               // Sinal de andon do posto 6
           ELSIF #Out_LinhaEcu.Andons[5] THEN
               #Out_LinhaEcu.NumMensagem := 14;
               #Out_MensagemEcu := 'NECESSARIO AJUDA NO POSTO 6';

               // Sinal de andon do posto 7
           ELSIF #Out_LinhaEcu.Andons[6] THEN
               #Out_LinhaEcu.NumMensagem := 15;
               #Out_MensagemEcu := 'NECESSARIO AJUDA NO POSTO 7';

               // Sinal de andon do posto 8
           ELSIF #Out_LinhaEcu.Andons[7] THEN
               #Out_LinhaEcu.NumMensagem := 16;
               #Out_MensagemEcu := 'AGUARDANDO RETIRADA DO PRODUTO NO POSTO 8';

           END_IF;
           ;
           // Linha em parada de produção
       ELSIF #S_ForaDeTurno THEN
           #Out_LinhaEcu.NumMensagem := 17;
           #Out_MensagemEcu := 'LINHA EM PARADA DE PRODUÇÃO';

           // Verifica se o AGV está em modo manual
       ELSIF (#In_DadosEcu.Dados_Agv[0].AutomaticoManual = 1) OR
           (#In_DadosEcu.Dados_Agv[1].AutomaticoManual = 1) OR
           (#In_DadosEcu.Dados_Agv[2].AutomaticoManual = 1) OR
           (#In_DadosEcu.Dados_Agv[3].AutomaticoManual = 1) OR
             (#In_DadosEcu.Dados_Agv[4].AutomaticoManual = 1) OR
             (*(#In_DadosEcu.Dados_Agv[5].AutomaticoManual = 1) OR*)
           (#In_DadosEcu.Dados_Agv[6].AutomaticoManual = 1) OR 
           (#In_DadosEcu.Dados_Agv[7].AutomaticoManual = 1) THEN

           // Verifica se o AGV 1 está em modo manual e diz em qual posto
           IF (#In_DadosEcu.Dados_Agv[0].AutomaticoManual = 1) THEN
               #Out_LinhaEcu.NumMensagem := 18;
               #Out_MensagemEcu := CONCAT(IN1 := 'AGV 1 EM MODO MANUAL NO POSTO ', IN2 := INT_TO_STRING(#In_DadosEcu.Dados_Agv[0].Posto));

               // Verifica se o AGV 2 está em modo manual e diz em qual posto
           ELSIF (#In_DadosEcu.Dados_Agv[1].AutomaticoManual = 1) THEN
               #Out_LinhaEcu.NumMensagem := 19;
               #Out_MensagemEcu := CONCAT(IN1 := 'AGV 2  EM MODO MANUAL NO POSTO ', IN2 := INT_TO_STRING(#In_DadosEcu.Dados_Agv[1].Posto));

               // Verifica se o AGV 3 está em modo manual e diz em qual posto
           ELSIF (#In_DadosEcu.Dados_Agv[2].AutomaticoManual = 1) THEN
               #Out_LinhaEcu.NumMensagem := 20;
               #Out_MensagemEcu := CONCAT(IN1 := 'AGV 3 EM MODO MANUAL NO POSTO ', IN2 := INT_TO_STRING(#In_DadosEcu.Dados_Agv[2].Posto));

               // Verifica se o AGV 4 está em modo manual e diz em qual posto
           ELSIF (#In_DadosEcu.Dados_Agv[3].AutomaticoManual = 1) THEN
               #Out_LinhaEcu.NumMensagem := 21;
               #Out_MensagemEcu := CONCAT(IN1 := 'AGV 4 EM MODO MANUAL NO POSTO ', IN2 := INT_TO_STRING(#In_DadosEcu.Dados_Agv[3].Posto));

               // Verifica se o AGV 5 está em modo manual e diz em qual posto
           ELSIF (#In_DadosEcu.Dados_Agv[4].AutomaticoManual = 1 AND "AlwaysFALSE") THEN
               #Out_LinhaEcu.NumMensagem := 22;
               #Out_MensagemEcu := CONCAT(IN1 := 'AGV 5 EM MODO MANUAL NO POSTO ', IN2 := INT_TO_STRING(#In_DadosEcu.Dados_Agv[4].Posto));

               // Verifica se o AGV 6 está em modo manual e diz em qual posto
               (* ELSIF (#In_DadosEcu.Dados_Agv[5].AutomaticoManual = 1 AND "AlwaysFALSE") THEN
               #Out_LinhaEcu.NumMensagem := 23;
               #Out_MensagemEcu := CONCAT(IN1 := 'AGV 6 EM MODO MANUAL NO POSTO ', IN2 := INT_TO_STRING(#In_DadosEcu.Dados_Agv[5].Posto));
               *)
               // Verifica se o AGV 7 está em modo manual e diz em qual posto
           ELSIF (#In_DadosEcu.Dados_Agv[6].AutomaticoManual = 1) THEN
               #Out_LinhaEcu.NumMensagem := 24;
               #Out_MensagemEcu := CONCAT(IN1 := 'AGV 7 EM MODO MANUAL NO POSTO ', IN2 := INT_TO_STRING(#In_DadosEcu.Dados_Agv[6].Posto));

               // Verifica se o AGV 8 está em modo manual e diz em qual posto
           ELSIF (#In_DadosEcu.Dados_Agv[7].AutomaticoManual = 1) THEN
               #Out_LinhaEcu.NumMensagem := 25;
               #Out_MensagemEcu := CONCAT(IN1 := 'AGV8 EM MODO MANUAL NO POSTO ', IN2 := INT_TO_STRING(#In_DadosEcu.Dados_Agv[7].Posto));


           END_IF;


           //Verifica se algum AGV esta fora da rota
       ELSIF (#In_DadosEcu.Dados_Agv[0]."Erros.Agv"= 8) OR
           (#In_DadosEcu.Dados_Agv[1]."Erros.Agv" = 8) OR
           (#In_DadosEcu.Dados_Agv[2]."Erros.Agv" = 8) OR
           (#In_DadosEcu.Dados_Agv[3]."Erros.Agv" = 8) OR
           (#In_DadosEcu.Dados_Agv[4]."Erros.Agv" = 8 ) OR
           (#In_DadosEcu.Dados_Agv[5]."Erros.Agv" = 8 AND "AlwaysFALSE") OR
           (#In_DadosEcu.Dados_Agv[6]."Erros.Agv" = 8) OR
           (#In_DadosEcu.Dados_Agv[7]."Erros.Agv" = 8) THEN

           // Verifica se o AGV 1 está fora da rota
           IF (#In_DadosEcu.Dados_Agv[0]."Erros.Pgv" = 8) THEN
               #Out_LinhaEcu.NumMensagem := 26;
               #Out_MensagemEcu := CONCAT(IN1 := 'AGV 1 FORA DA ROTA NO POSTO ', IN2 := INT_TO_STRING(#In_DadosEcu.Dados_Agv[0].Posto));

               // Verifica se o AGV 2 está fora da rota
           ELSIF (#In_DadosEcu.Dados_Agv[1]."Erros.Agv" = 8) THEN
               #Out_LinhaEcu.NumMensagem := 27;
               #Out_MensagemEcu := CONCAT(IN1 := 'AGV 2 FORA DA ROTA NO POSTO ', IN2 := INT_TO_STRING(#In_DadosEcu.Dados_Agv[1].Posto));

               // Verifica se o AGV 3 está fora da rota
           ELSIF (#In_DadosEcu.Dados_Agv[2]."Erros.Agv" = 8) THEN
               #Out_LinhaEcu.NumMensagem := 28;
               #Out_MensagemEcu := CONCAT(IN1 := 'AGV 3 FORA DA ROTA NO POSTO ', IN2 := INT_TO_STRING(#In_DadosEcu.Dados_Agv[2].Posto));

               // Verifica se o AGV 4 está fora da rota
           ELSIF (#In_DadosEcu.Dados_Agv[3]."Erros.Agv" = 8) THEN
               #Out_LinhaEcu.NumMensagem := 29;
               #Out_MensagemEcu := CONCAT(IN1 := 'AGV 4 FORA DA ROTA NO POSTO ', IN2 := INT_TO_STRING(#In_DadosEcu.Dados_Agv[3].Posto));

               // Verifica se o AGV 5 está fora da rota
           ELSIF (#In_DadosEcu.Dados_Agv[4]."Erros.Agv" = 8 AND "AlwaysFALSE") THEN
               #Out_LinhaEcu.NumMensagem := 30;
               #Out_MensagemEcu := CONCAT(IN1 := 'AGV 5 FORA DA ROTA NO POSTO ', IN2 := INT_TO_STRING(#In_DadosEcu.Dados_Agv[4].Posto));

               // Verifica se o AGV 6 está fora da rota
           ELSIF (#In_DadosEcu.Dados_Agv[5]."Erros.Agv" = 8 AND "AlwaysFALSE") THEN
               #Out_LinhaEcu.NumMensagem := 31;
               #Out_MensagemEcu := CONCAT(IN1 := 'AGV 6 FORA DA ROTA NO POSTO ', IN2 := INT_TO_STRING(#In_DadosEcu.Dados_Agv[5].Posto));
               // Verifica se o AGV 7 está fora da rota
           ELSIF (#In_DadosEcu.Dados_Agv[6]."Erros.Agv" = 8) THEN
               #Out_LinhaEcu.NumMensagem := 32;
               #Out_MensagemEcu := CONCAT(IN1 := 'AGV 7 FORA DA ROTA NO POSTO ', IN2 := INT_TO_STRING(#In_DadosEcu.Dados_Agv[6].Posto));
               // Verifica se o AGV 8 está fora da rota
           ELSIF (#In_DadosEcu.Dados_Agv[7]."Erros.Agv" = 8) THEN
               #Out_LinhaEcu.NumMensagem := 33;
               #Out_MensagemEcu := CONCAT(IN1 := 'AGV 8 FORA DA ROTA NO POSTO ', IN2 := INT_TO_STRING(#In_DadosEcu.Dados_Agv[7].Posto));


           END_IF; 

       ELSE
           #Out_LinhaEcu.NumMensagem := 0;
           #Out_MensagemEcu := 'LINHA LIBERADA';
       END_IF;

   END_REGION

   // Coloca os dados das memorias nas saidas do bloco
   REGION Saidas
       // Coloca os dados das memorias nas saidas do bloco
       #Out_LinhaEcu.Tempo_Takt := #In_DadosEcu.Dados_Takt.Tempo_Takt;
       #Out_LinhaEcu.Tempo_StopTime := #In_DadosEcu.Dados_Takt.Tempo_StopTime;
       #Out_LinhaEcu.Objetivo := #In_DadosEcu.Dados_Takt.Objetivo;
       #Out_LinhaEcu.Atual := #In_DadosEcu.Dados_Takt.Atual;
       #Out_LinhaEcu.DirectRun := 99.9;
       #Out_LinhaEcu.LinhaParada := #S_ForaDeTurno;
       #Out_LinhaEcu.TempoRetornoParada := #S_TempoRetorno;
       #Out_LinhaEcu.LinhaRodando := NOT #S_ForaDeTurno;
   END_REGION
END_FUNCTION_BLOCK

FUNCTION_BLOCK "FB203_FiltroDados_Skd"   // FB203, SCL
TITLE = FB203_FiltroDados_Skd
{ S7_Optimized_Access := 'TRUE' }
VERSION : 0.1
// FB203_FiltroDados_Skd
   VAR_INPUT
      In_InfoCabinas : "TAKT_OUTPUT.INFORMATION";
      In_Turno : Struct
         Turnos : Array[0..2] of Struct
            Inicio : Date_And_Time;
            Fim : Date_And_Time;
            Objetivo : Int;
            DiasDaSemana : Array[0..6] of Bool;
            Paradas : Array[0..5] of Struct
               Inicio : Date_And_Time;
               Fim : Date_And_Time;
            END_STRUCT;
            HE_Inicio : Date_And_Time;
            HE_Fim : Date_And_Time;
         END_STRUCT;
      END_STRUCT;
   END_VAR
   VAR_OUTPUT
      Out_Linha : Struct
         Tempo_Takt : DInt;
         Tempo_StopTime : DInt;
         Objetivo : Int;
         Atual : Int;
         LinhaParada : Bool;
         TempoRetornoParada : DInt;
         LinhaRodando : Bool;
         Andons : Array[0..8] of Bool;
         CorDeTela : Byte;
         DirectRun : Real;
         SaldoDoTurno : Int;
         AndonOn : Int;
         Paradas : Array[0..1] of Struct
            Inicio : Time_Of_Day;
            Fim : Time_Of_Day;
            Posto : Int;
            ValorTimer : Int;
            ValorTimerFim : Int;
         END_STRUCT;
         NumMensagem : Int;
         Emergencias : Array[0..8] of Bool;
      END_STRUCT;
      Out_Mensagem : String;
   END_VAR
   VAR
      S_DateTime : Date_And_Time;
      S_CounterFor : Int;
      S_CounterFor_1 : Int;
      S_Turnos : Array[0..2] of Struct
         Paradas : Array[0..6] of Bool;
         ContagemRetorno : Array[0..6] of DInt;
      END_STRUCT;
      S_ForaDeTurno : Bool;
      S_TempoRetorno : DInt;
      S_Hora : Time_Of_Day;
   END_VAR
   VAR_TEMP
      Err : Int;
   END_VAR
BEGIN
   (*
       ESTE BLOCO REALIZA O FILTRO DAS INFORMAÇÕES DO TAKT, EXEMPLOS: TROCA DA COR DA TELA, MENSAGENS NA TELA E ETC
   *)


   // Converte o sinal de andon de byte para boolean
   REGION Valores ANDON
       // Converte o sinal de andon de byte para boolean
       #Out_Linha.Andons[0] := #In_InfoCabinas.ANDON.%X0;
       #Out_Linha.Andons[1] := #In_InfoCabinas.ANDON.%X1;
       #Out_Linha.Andons[2] := #In_InfoCabinas.ANDON.%X2;
       #Out_Linha.Andons[3] := #In_InfoCabinas.ANDON.%X3;
       #Out_Linha.Andons[4] := #In_InfoCabinas.ANDON.%X4;
       #Out_Linha.Andons[5] := #In_InfoCabinas.ANDON.%X5;
       #Out_Linha.Andons[6] := #In_InfoCabinas.ANDON.%X6;
       #Out_Linha.Andons[7] := #In_InfoCabinas.ANDON.%X7;
   END_REGION

   // Converte o sinal de emergencia de byte para boolean
   REGION Valores Emergencia
       // Converte o sinal de emergencia de byte para boolean
       #Out_Linha.Emergencias[0] := #In_InfoCabinas.EMERGENCY.%X0;
       #Out_Linha.Emergencias[1] := #In_InfoCabinas.EMERGENCY.%X1;
       #Out_Linha.Emergencias[2] := #In_InfoCabinas.EMERGENCY.%X2;
       #Out_Linha.Emergencias[3] := #In_InfoCabinas.EMERGENCY.%X3;
       #Out_Linha.Emergencias[4] := #In_InfoCabinas.EMERGENCY.%X4;
       #Out_Linha.Emergencias[5] := #In_InfoCabinas.EMERGENCY.%X5;
       #Out_Linha.Emergencias[6] := #In_InfoCabinas.EMERGENCY.%X6;
       #Out_Linha.Emergencias[7] := #In_InfoCabinas.EMERGENCY.%X7;
   END_REGION

   //Realiza a leitura da hora atual do CLP
   REGION HoraAtual

       //Realiza a leitura da hora atual do CLP
       #Err := RD_LOC_T(#S_DateTime);

   END_REGION
   REGION VerificaEmTurno
       #S_Hora := DT_TO_TOD(#S_DateTime);
       IF #S_Hora > TOD#16:00:00 THEN
           #S_TempoRetorno := TOD_TO_DINT(TOD#07:00:00) - TOD_TO_DINT(#S_Hora);
           #S_ForaDeTurno := 1;
       ELSE
           #S_TempoRetorno := 0;
           #S_ForaDeTurno := 0;
       END_IF;


   END_REGION
   //Verifica se a linha esta em turno, caso não esteja retorno o tempo necessario para a linha voltar a rodar
   REGION LinhaEmTurno
       FOR #S_CounterFor := 0 TO 2 DO
           //Verifica se está em turno
           IF #In_Turno.Turnos[#S_CounterFor].Inicio >= #S_DateTime AND #S_DateTime <= #In_Turno.Turnos[#S_CounterFor].Fim THEN
               //Verifica se existe alguma parada programada
               FOR #S_CounterFor_1 := 0 TO 5 DO
                   IF #In_Turno.Turnos[#S_CounterFor].Paradas[#S_CounterFor_1].Inicio >= #S_DateTime
                       AND #S_DateTime <= #In_Turno.Turnos[#S_CounterFor].Paradas[#S_CounterFor_1].Fim THEN

                       #S_Turnos[#S_CounterFor].Paradas[#S_CounterFor_1] := 1;
                       #S_Turnos[#S_CounterFor].ContagemRetorno[#S_CounterFor_1] := TOD_TO_DINT(DT_TO_TOD(#S_DateTime - (#In_Turno.Turnos[#S_CounterFor].Paradas[#S_CounterFor_1].Fim - #In_Turno.Turnos[#S_CounterFor].Paradas[#S_CounterFor_1].Inicio)));
                   ELSE
                       #S_Turnos[#S_CounterFor].ContagemRetorno[#S_CounterFor_1] := 0;
                       #S_Turnos[#S_CounterFor].Paradas[#S_CounterFor_1] := 0;

                   END_IF;

                   #S_Turnos[#S_CounterFor].Paradas[6] := 0; // Em turno
                   #S_Turnos[#S_CounterFor].ContagemRetorno[6] := 0;
               END_FOR;
           ELSE
               #S_Turnos[#S_CounterFor].Paradas[6] := 1; // Fora de turno
               #S_Turnos[#S_CounterFor].ContagemRetorno[6] := #S_DateTime - #In_Turno.Turnos[#S_CounterFor].Paradas[#S_CounterFor_1].Inicio; // Quantidade de tempo restante para reiniciar o novo turno
           END_IF;

       END_FOR;

       #S_ForaDeTurno := #S_Turnos[0 AND 1 AND 2].Paradas[0 AND 1 AND 2 AND 3 AND 4 AND 5 AND 6];
       #S_TempoRetorno := #S_Turnos[0 AND 1 AND 2].ContagemRetorno[0 AND 1 AND 2 AND 3 AND 4 AND 5 AND 6];
   END_REGION

   // Realiza a analise de todos os dados e troca a cor da tela
   REGION DefiniçãoCorDaTela
       // 1 - Tela Amarela (Necessario ajuda em algum posto e não estourou o tempo do TAKT)
       IF ((#Out_Linha.Andons[1] OR #Out_Linha.Andons[3] OR #Out_Linha.Andons[4] OR #Out_Linha.Andons[6] OR #Out_Linha.Andons[7]) AND (#In_InfoCabinas.TAKT_ET > 0) AND NOT #S_ForaDeTurno) THEN
           #Out_Linha.CorDeTela := 1;

           // 2 - Tela Vermelho (Necessario ajuda em algum posto e estourou o tempo do TAKT)
       ELSIF (((#Out_Linha.Andons[0] OR #Out_Linha.Andons[1] OR #Out_Linha.Andons[3] OR #Out_Linha.Andons[4] OR #Out_Linha.Andons[6] OR #Out_Linha.Andons[7]) AND (#In_InfoCabinas.TAKT_ET = 0)) OR (#In_InfoCabinas.EMERGENCY <> 0)) AND NOT #S_ForaDeTurno THEN
           #Out_Linha.CorDeTela := 2;

           //3 - Tela Azul - (Aguardando inicio de turno/Volta da refeição)
       ELSIF #S_ForaDeTurno THEN
           #Out_Linha.CorDeTela := 3;

           //4 - Tela Laranja - (Aguardando retirada do produto)
       ELSIF ((#Out_Linha.Andons[0] OR #Out_Linha.Andons[7])) AND NOT #S_ForaDeTurno THEN
           #Out_Linha.CorDeTela := 4;
           //0 - Tela Branca/Preta (Tudo Ok)
       ELSE
           #Out_Linha.CorDeTela := 0;
       END_IF;


   END_REGION

   // Realiza a analise de todos os dados e escreve a mensagem na tela 
   REGION Mensagens

       IF #In_InfoCabinas.EMERGENCY <> 0 AND NOT #S_ForaDeTurno THEN

           // Sinal de EMERGÊNCIA  do posto 1
           IF #Out_Linha.Emergencias[0] THEN
               #Out_Linha.NumMensagem := 1;
               #Out_Mensagem := 'EMERGÊNCIA  ACIONADO NO POSTO 1';

               // Sinal de EMERGÊNCIA  do posto 2
           ELSIF #Out_Linha.Emergencias[1] THEN
               #Out_Linha.NumMensagem := 2;
               #Out_Mensagem := 'EMERGÊNCIA  ACIONADO NO POSTO 2';

               // Sinal de EMERGÊNCIA  do posto 3
           ELSIF #Out_Linha.Emergencias[2] THEN
               #Out_Linha.NumMensagem := 3;
               #Out_Mensagem := 'EMERGÊNCIA  ACIONADO NO POSTO 3';

               // Sinal de EMERGÊNCIA  do posto 4
           ELSIF #Out_Linha.Emergencias[3] THEN
               #Out_Linha.NumMensagem := 4;
               #Out_Mensagem := 'EMERGÊNCIA  ACIONADO NO POSTO 4';

               // Sinal de EMERGÊNCIA  do posto 5
           ELSIF #Out_Linha.Emergencias[4] THEN
               #Out_Linha.NumMensagem := 5;
               #Out_Mensagem := 'EMERGÊNCIA  ACIONADO NO POSTO 5';

               // Sinal de EMERGÊNCIA  do posto 6
           ELSIF #Out_Linha.Emergencias[5] THEN
               #Out_Linha.NumMensagem := 6;
               #Out_Mensagem := 'EMERGÊNCIA  ACIONADO NO POSTO 6';

               // Sinal de EMERGÊNCIA  do posto 7
           ELSIF #Out_Linha.Emergencias[6] THEN
               #Out_Linha.NumMensagem := 7;
               #Out_Mensagem := 'EMERGÊNCIA  ACIONADO NO POSTO 7';

               // Sinal de EMERGÊNCIA  do posto 8
           ELSIF #Out_Linha.Emergencias[7] THEN
               #Out_Linha.NumMensagem := 8;
               #Out_Mensagem := 'EMERGÊNCIA  ACIONADO NO POSTO 8';

           END_IF;

       ELSIF #In_InfoCabinas.ANDON <> 0 AND NOT #S_ForaDeTurno THEN

           // Sinal de andon do posto 1
           IF #Out_Linha.Andons[0] THEN
               #Out_Linha.NumMensagem := 9;
               #Out_Mensagem := 'NECESSARIO AJUDA NO POSTO 1';

               // Sinal de andon do posto 2
           ELSIF #Out_Linha.Andons[1] THEN
               #Out_Linha.NumMensagem := 10;
               #Out_Mensagem := 'NECESSARIO AJUDA NO POSTO 2';

               // Sinal de andon do posto 3
           ELSIF #Out_Linha.Andons[2] THEN
               #Out_Linha.NumMensagem := 11;
               #Out_Mensagem := 'NECESSARIO AJUDA NO POSTO 3';

               // Sinal de andon do posto 4
           ELSIF #Out_Linha.Andons[3] THEN
               #Out_Linha.NumMensagem := 12;
               #Out_Mensagem := 'NECESSARIO AJUDA NO POSTO 4';

               // Sinal de andon do posto 5
           ELSIF #Out_Linha.Andons[4] THEN
               #Out_Linha.NumMensagem := 13;
               #Out_Mensagem := 'NECESSARIO AJUDA NO POSTO 5';

               // Sinal de andon do posto 6
           ELSIF #Out_Linha.Andons[5] THEN
               #Out_Linha.NumMensagem := 14;
               #Out_Mensagem := 'NECESSARIO AJUDA NO POSTO 6';

               // Sinal de andon do posto 7
           ELSIF #Out_Linha.Andons[6] THEN
               #Out_Linha.NumMensagem := 15;
               #Out_Mensagem := 'NECESSARIO AJUDA NO POSTO 7';

               // Sinal de andon do posto 8
           ELSIF #Out_Linha.Andons[7] THEN
               #Out_Linha.NumMensagem := 16;
               #Out_Mensagem := 'NECESSARIO AJUDA NO POSTO 8';

           END_IF;
           ;
           // Linha em parada de produção
       ELSIF #S_ForaDeTurno THEN
           #Out_Linha.NumMensagem := 17;
           #Out_Mensagem := 'LINHA EM PARADA DE PRODUÇÃO';
       ELSE
           #Out_Linha.NumMensagem := 0;
           #Out_Mensagem := 'LINHA LIBERADA';
       END_IF;

   END_REGION

   // Coloca os dados das memorias nas saidas do bloco
   REGION Saidas
       // Coloca os dados das memorias nas saidas do bloco
       #Out_Linha.Tempo_Takt := #In_InfoCabinas.TAKT_ET;
       #Out_Linha.Tempo_StopTime := #In_InfoCabinas.STOP_TIME;
       #Out_Linha.Objetivo := #In_InfoCabinas.TARGET;
       #Out_Linha.Atual := #In_InfoCabinas.ACTUAL_PRODUCTION;
       #Out_Linha.DirectRun := 99.9;
       #Out_Linha.LinhaParada := #S_ForaDeTurno;
       #Out_Linha.TempoRetornoParada := #S_TempoRetorno;
       #Out_Linha.LinhaRodando := NOT #S_ForaDeTurno;
   END_REGION
END_FUNCTION_BLOCK

FUNCTION_BLOCK "FB204_FiltroDados_Comp"   // FB204, SCL
TITLE = FB204_FiltroDados_Comp
{ S7_Optimized_Access := 'TRUE' }
VERSION : 0.1
// FB204_FiltroDados_Comp
   VAR_INPUT
      In_InfoCabinas : "TAKT_OUTPUT.INFORMATION";
      In_Turno : Struct
         Turnos : Array[0..2] of Struct
            Inicio : Date_And_Time;
            Fim : Date_And_Time;
            Objetivo : Int;
            DiasDaSemana : Array[0..6] of Bool;
            Paradas : Array[0..5] of Struct
               Inicio : Date_And_Time;
               Fim : Date_And_Time;
            END_STRUCT;
            HE_Inicio : Date_And_Time;
            HE_Fim : Date_And_Time;
         END_STRUCT;
      END_STRUCT;
   END_VAR
   VAR_OUTPUT
      Out_Linha : Struct
         Tempo_Takt : DInt;
         Tempo_StopTime : DInt;
         Objetivo : Int;
         Atual : Int;
         LinhaParada : Bool;
         TempoRetornoParada : DInt;
         LinhaRodando : Bool;
         Andons : Array[0..8] of Bool;
         CorDeTela : Byte;
         DirectRun : Real;
         SaldoDoTurno : Int;
         AndonOn : Int;
         Paradas : Array[0..1] of Struct
            Inicio : Time_Of_Day;
            Fim : Time_Of_Day;
            Posto : Int;
            ValorTimer : Int;
            ValorTimerFim : Int;
         END_STRUCT;
         NumMensagem : Int;
         Emergencias : Array[0..8] of Bool;
      END_STRUCT;
      Out_Mensagem : String;
   END_VAR
   VAR
      S_DateTime : Date_And_Time;
      S_CounterFor : Int;
      S_CounterFor_1 : Int;
      S_Turnos : Array[0..2] of Struct
         Paradas : Array[0..6] of Bool;
         ContagemRetorno : Array[0..6] of DInt;
      END_STRUCT;
      S_ForaDeTurno : Bool;
      S_TempoRetorno : DInt;
      S_Hora : Time_Of_Day;
   END_VAR
   VAR_TEMP
      Err : Int;
   END_VAR
BEGIN
   (*
       ESTE BLOCO REALIZA O FILTRO DAS INFORMAÇÕES DO TAKT, EXEMPLOS: TROCA DA COR DA TELA, MENSAGENS NA TELA E ETC
   *)


   // Converte o sinal de andon de byte para boolean
   REGION Valores ANDON
       // Converte o sinal de andon de byte para boolean
       #Out_Linha.Andons[0] := #In_InfoCabinas.ANDON.%X0;
       #Out_Linha.Andons[1] := #In_InfoCabinas.ANDON.%X1;
       #Out_Linha.Andons[2] := #In_InfoCabinas.ANDON.%X2;
       #Out_Linha.Andons[3] := #In_InfoCabinas.ANDON.%X3;
       #Out_Linha.Andons[4] := #In_InfoCabinas.ANDON.%X4;
       #Out_Linha.Andons[5] := #In_InfoCabinas.ANDON.%X5;
       #Out_Linha.Andons[6] := #In_InfoCabinas.ANDON.%X6;
       #Out_Linha.Andons[7] := #In_InfoCabinas.ANDON.%X7;
   END_REGION

   // Converte o sinal de emergencia de byte para boolean
   REGION Valores Emergencia
       // Converte o sinal de emergencia de byte para boolean
       #Out_Linha.Emergencias[0] := #In_InfoCabinas.EMERGENCY.%X0;
       #Out_Linha.Emergencias[1] := #In_InfoCabinas.EMERGENCY.%X1;
       #Out_Linha.Emergencias[2] := #In_InfoCabinas.EMERGENCY.%X2;
       #Out_Linha.Emergencias[3] := #In_InfoCabinas.EMERGENCY.%X3;
       #Out_Linha.Emergencias[4] := #In_InfoCabinas.EMERGENCY.%X4;
       #Out_Linha.Emergencias[5] := #In_InfoCabinas.EMERGENCY.%X5;
       #Out_Linha.Emergencias[6] := #In_InfoCabinas.EMERGENCY.%X6;
       #Out_Linha.Emergencias[7] := #In_InfoCabinas.EMERGENCY.%X7;
   END_REGION

   //Realiza a leitura da hora atual do CLP
   REGION HoraAtual

       //Realiza a leitura da hora atual do CLP
       #Err := RD_LOC_T(#S_DateTime);

   END_REGION
   REGION VerificaEmTurno
       #S_Hora := DT_TO_TOD(#S_DateTime);
       IF #S_Hora > TOD#16:00:00 THEN
           #S_TempoRetorno := TOD_TO_DINT(TOD#07:00:00) - TOD_TO_DINT(#S_Hora);
           #S_ForaDeTurno := 1;
       ELSE
           #S_TempoRetorno := 0;
           #S_ForaDeTurno := 0;
       END_IF;


   END_REGION
   //Verifica se a linha esta em turno, caso não esteja retorno o tempo necessario para a linha voltar a rodar
   REGION LinhaEmTurno
       FOR #S_CounterFor := 0 TO 2 DO
           //Verifica se está em turno
           IF #In_Turno.Turnos[#S_CounterFor].Inicio >= #S_DateTime AND #S_DateTime <= #In_Turno.Turnos[#S_CounterFor].Fim THEN
               //Verifica se existe alguma parada programada
               FOR #S_CounterFor_1 := 0 TO 5 DO
                   IF #In_Turno.Turnos[#S_CounterFor].Paradas[#S_CounterFor_1].Inicio >= #S_DateTime
                       AND #S_DateTime <= #In_Turno.Turnos[#S_CounterFor].Paradas[#S_CounterFor_1].Fim THEN

                       #S_Turnos[#S_CounterFor].Paradas[#S_CounterFor_1] := 1;
                       #S_Turnos[#S_CounterFor].ContagemRetorno[#S_CounterFor_1] := TOD_TO_DINT(DT_TO_TOD(#S_DateTime - (#In_Turno.Turnos[#S_CounterFor].Paradas[#S_CounterFor_1].Fim - #In_Turno.Turnos[#S_CounterFor].Paradas[#S_CounterFor_1].Inicio)));
                   ELSE
                       #S_Turnos[#S_CounterFor].ContagemRetorno[#S_CounterFor_1] := 0;
                       #S_Turnos[#S_CounterFor].Paradas[#S_CounterFor_1] := 0;

                   END_IF;

                   #S_Turnos[#S_CounterFor].Paradas[6] := 0; // Em turno
                   #S_Turnos[#S_CounterFor].ContagemRetorno[6] := 0;
               END_FOR;
           ELSE
               #S_Turnos[#S_CounterFor].Paradas[6] := 1; // Fora de turno
               #S_Turnos[#S_CounterFor].ContagemRetorno[6] := #S_DateTime - #In_Turno.Turnos[#S_CounterFor].Paradas[#S_CounterFor_1].Inicio; // Quantidade de tempo restante para reiniciar o novo turno
           END_IF;

       END_FOR;

       #S_ForaDeTurno := #S_Turnos[0 AND 1 AND 2].Paradas[0 AND 1 AND 2 AND 3 AND 4 AND 5 AND 6];
       #S_TempoRetorno := #S_Turnos[0 AND 1 AND 2].ContagemRetorno[0 AND 1 AND 2 AND 3 AND 4 AND 5 AND 6];
   END_REGION

   // Realiza a analise de todos os dados e troca a cor da tela
   REGION DefiniçãoCorDaTela
       // 1 - Tela Amarela (Necessario ajuda em algum posto e não estourou o tempo do TAKT)
       IF (( #Out_Linha.Andons[1] OR #Out_Linha.Andons[3] OR #Out_Linha.Andons[5] OR #Out_Linha.Andons[7]) AND (#In_InfoCabinas.TAKT_ET > 0)) AND NOT #S_ForaDeTurno THEN
           #Out_Linha.CorDeTela := 1;

           // 2 - Tela Vermelho (Necessario ajuda em algum posto e estourou o tempo do TAKT)
       ELSIF ((( #Out_Linha.Andons[1] OR #Out_Linha.Andons[3] OR #Out_Linha.Andons[5] OR #Out_Linha.Andons[7]) AND (#In_InfoCabinas.TAKT_ET <= 0)) OR (#In_InfoCabinas.EMERGENCY <> 0)) AND NOT #S_ForaDeTurno THEN
           #Out_Linha.CorDeTela := 2;

           //3 - Tela Azul - (Aguardando inicio de turno/Volta da refeição)
       ELSIF #S_ForaDeTurno THEN
           #Out_Linha.CorDeTela := 3;

           //4 - Tela Laranja - (Aguardando retirada do produto)
       ELSIF ((#Out_Linha.Andons[0] OR #Out_Linha.Andons[4])) AND NOT #S_ForaDeTurno THEN
           #Out_Linha.CorDeTela := 4;
           //0 - Tela Branca/Preta (Tudo Ok)
       ELSE
           #Out_Linha.CorDeTela := 0;
       END_IF;


   END_REGION

   // Realiza a analise de todos os dados e escreve a mensagem na tela 
   REGION Mensagens

       IF #In_InfoCabinas.EMERGENCY <> 0 AND NOT #S_ForaDeTurno THEN

           // Sinal de EMERGÊNCIA  do posto 1
           IF #Out_Linha.Emergencias[0] THEN
               #Out_Linha.NumMensagem := 1;
               #Out_Mensagem := 'EMERGÊNCIA  ACIONADO NO POSTO 1';

               // Sinal de EMERGÊNCIA  do posto 2
           ELSIF #Out_Linha.Emergencias[1] THEN
               #Out_Linha.NumMensagem := 2;
               #Out_Mensagem := 'EMERGÊNCIA  ACIONADO NO POSTO 2';

               // Sinal de EMERGÊNCIA  do posto 3
           ELSIF #Out_Linha.Emergencias[2] THEN
               #Out_Linha.NumMensagem := 3;
               #Out_Mensagem := 'EMERGÊNCIA  ACIONADO NO POSTO 3';

               // Sinal de EMERGÊNCIA  do posto 4
           ELSIF #Out_Linha.Emergencias[3] THEN
               #Out_Linha.NumMensagem := 4;
               #Out_Mensagem := 'EMERGÊNCIA  ACIONADO NO POSTO 4';

               // Sinal de EMERGÊNCIA  do posto 5
           ELSIF #Out_Linha.Emergencias[4] THEN
               #Out_Linha.NumMensagem := 5;
               #Out_Mensagem := 'EMERGÊNCIA  ACIONADO NO POSTO 5';

               // Sinal de EMERGÊNCIA  do posto 6
           ELSIF #Out_Linha.Emergencias[5] THEN
               #Out_Linha.NumMensagem := 6;
               #Out_Mensagem := 'EMERGÊNCIA  ACIONADO NO POSTO 6';

               // Sinal de EMERGÊNCIA  do posto 7
           ELSIF #Out_Linha.Emergencias[6] THEN
               #Out_Linha.NumMensagem := 7;
               #Out_Mensagem := 'EMERGÊNCIA  ACIONADO NO POSTO 7';

               // Sinal de EMERGÊNCIA  do posto 8
           ELSIF #Out_Linha.Emergencias[7] THEN
               #Out_Linha.NumMensagem := 8;
               #Out_Mensagem := 'EMERGÊNCIA  ACIONADO NO POSTO 8';

           END_IF;

       ELSIF #In_InfoCabinas.ANDON <> 0 AND NOT #S_ForaDeTurno THEN

           // Sinal de andon do posto 1
           IF #Out_Linha.Andons[0] THEN
               #Out_Linha.NumMensagem := 9;
               #Out_Mensagem := 'NECESSARIO AJUDA NO POSTO 1';

               // Sinal de andon do posto 2
           ELSIF #Out_Linha.Andons[1] THEN
               #Out_Linha.NumMensagem := 10;
               #Out_Mensagem := 'NECESSARIO AJUDA NO POSTO 2';

               // Sinal de andon do posto 3
           ELSIF #Out_Linha.Andons[2] THEN
               #Out_Linha.NumMensagem := 11;
               #Out_Mensagem := 'NECESSARIO AJUDA NO POSTO 3';

               // Sinal de andon do posto 4
           ELSIF #Out_Linha.Andons[3] THEN
               #Out_Linha.NumMensagem := 12;
               #Out_Mensagem := 'NECESSARIO AJUDA NO POSTO 4';

               // Sinal de andon do posto 5
           ELSIF #Out_Linha.Andons[4] THEN
               #Out_Linha.NumMensagem := 13;
               #Out_Mensagem := 'AGUARDANDO RETIRADA DO PRODUTO NO POSTO 5';

               // Sinal de andon do posto 6
           ELSIF #Out_Linha.Andons[5] THEN
               #Out_Linha.NumMensagem := 14;
               #Out_Mensagem := 'NECESSARIO AJUDA NO POSTO 6';

               // Sinal de andon do posto 7
           ELSIF #Out_Linha.Andons[6] THEN
               #Out_Linha.NumMensagem := 15;
               #Out_Mensagem := 'NECESSARIO AJUDA NO POSTO 7';

               // Sinal de andon do posto 8
           ELSIF #Out_Linha.Andons[7] THEN
               #Out_Linha.NumMensagem := 16;
               #Out_Mensagem := 'NECESSARIO AJUDA NO POSTO 8';

           END_IF;
           ;
           // Linha em parada de produção
       ELSIF #S_ForaDeTurno THEN
           #Out_Linha.NumMensagem := 17;
           #Out_Mensagem := 'LINHA EM PARADA DE PRODUÇÃO';
       ELSE
           #Out_Linha.NumMensagem := 0;
           #Out_Mensagem := 'LINHA LIBERADA';
       END_IF;

   END_REGION

   // Coloca os dados das memorias nas saidas do bloco
   REGION Saidas
       // Coloca os dados das memorias nas saidas do bloco
       #Out_Linha.Tempo_Takt := #In_InfoCabinas.TAKT_ET;
       #Out_Linha.Tempo_StopTime := #In_InfoCabinas.STOP_TIME;
      #Out_Linha.Objetivo := #In_InfoCabinas.TARGET;
       #Out_Linha.Atual := #In_InfoCabinas.ACTUAL_PRODUCTION;
       #Out_Linha.DirectRun := 99.9;
       #Out_Linha.LinhaParada := #S_ForaDeTurno;
       #Out_Linha.TempoRetornoParada := #S_TempoRetorno;
       #Out_Linha.LinhaRodando := NOT #S_ForaDeTurno;
   END_REGION
END_FUNCTION_BLOCK

FUNCTION_BLOCK "FB205_FiltroDadosAgv"   // FB205, SCL
TITLE = FB205_FiltroDadosAgv
{ S7_Optimized_Access := 'TRUE' }
VERSION : 0.1
// FB205_FiltroDadosAgvs
   VAR_INPUT
      In : "Agv.Database";
   END_VAR
   VAR_OUTPUT
      Out_Sinais : Byte;
      Out_Posto : Byte;
      Out_Comando : Byte;
      Out_Velocidade : Byte;
      Out_Processo : Byte;
      Out_VelAtual : Byte;
      "Out_Erros.Agv" : Byte;
      "Out_Erros.Pgv" : Byte;
      "Out_Erros.MotorPasso" : Byte;
   END_VAR
BEGIN



   //#In_InfoCabinas.ANDON.%X0;
   IF #In.Emergencia THEN
       #Out_Sinais.%X0 := 1;
   ELSE
       #Out_Sinais.%X0 := 0;
   END_IF;

   IF #In.Safety THEN
       #Out_Sinais.%X1 := 1;
   ELSE
       #Out_Sinais.%X1 := 0;
   END_IF;

   IF #In.Warning THEN
       #Out_Sinais.%X2 := 1;
   ELSE
       #Out_Sinais.%X2 := 0;
   END_IF;

   IF #In.Rodando THEN
       #Out_Sinais.%X3 := 1;
   ELSE
       #Out_Sinais.%X3 := 0;
   END_IF;


   IF #In.AutomaticoManual = 2 THEN
       #Out_Sinais.%X4 := 1;
   ELSE
       #Out_Sinais.%X4 := 0;
   END_IF;

   IF #In.ConectarTakt  THEN
       #Out_Sinais.%X5 := 1;
   ELSE
       #Out_Sinais.%X5 := 0;
   END_IF;

   IF #In.Falha  THEN
       #Out_Sinais.%X6 := 1;
   ELSE
       #Out_Sinais.%X6 := 0;
   END_IF;

   IF #In.AutomaticoManual = 1 THEN
       #Out_Sinais.%X7 := 1;
   ELSE
       #Out_Sinais.%X7 := 0;
   END_IF;



   #Out_Posto := #In.Posto;
   #Out_Comando := #In.Comando;
   #Out_Velocidade := #In.Velocidade;
   #Out_Processo := #In.Processo;
   #Out_VelAtual := INT_TO_BYTE((#In.VelocidadeAtual/1000));
   #"Out_Erros.Agv" := #In."Erros.Agv";
   #"Out_Erros.Pgv" := #In."Erros.Pgv";
   #"Out_Erros.MotorPasso" := #In."Erros.Rfid";
END_FUNCTION_BLOCK

FUNCTION_BLOCK "FB206_CheckEmTurno"   // FB206, SCL
TITLE = FB206_EmTurno
{ S7_Optimized_Access := 'TRUE' }
VERSION : 0.1
   VAR_INPUT
      In_Turnos : Array[0..2] of Struct
         Inicio : Date_And_Time;
         Fim : Date_And_Time;
      END_STRUCT;
      In_Paradas : Array[0..5] of Struct
         Inicio : Time_Of_Day;
         Fim : Time_Of_Day;
      END_STRUCT;
   END_VAR
   VAR_OUTPUT
      Out_Parada : Bool;
      Out_TempoRetornoParada : Int;
      Out_EmDiaDeProd : Int;
   END_VAR
   VAR
      S_Index : Int;
      DateTime : Date_And_Time;
      TOD : Time_Of_Day;
      S_ForaDeTurno : Bool;
      S_TempoRetornoParada : Int;
      DTL : DTL;
   END_VAR
   VAR_TEMP
      Err : Int;
   END_VAR
BEGIN
   #Err := RD_LOC_T(#DTL);
   #Err := RD_SYS_T(#DateTime);
   #TOD := DTL_TO_TOD(#DTL);


   IF #In_Turnos[0].Fim > #DateTime THEN

       IF NOT (DTL_TO_TOD(#In_Turnos[1].Inicio) = TOD#00:00:00) THEN
           #S_ForaDeTurno := 1;
           #S_TempoRetornoParada := TOD_TO_INT((DTL_TO_TOD(#In_Turnos[1].Inicio))) - TOD_TO_INT(#TOD);
       ELSIF NOT (DTL_TO_TOD(#In_Turnos[2].Inicio) = TOD#00:00:00) THEN
           #S_ForaDeTurno := 1;
           #S_TempoRetornoParada := TOD_TO_INT((DTL_TO_TOD(#In_Turnos[2].Inicio))) - TOD_TO_INT(#TOD);
       ELSIF NOT (DTL_TO_TOD(#In_Turnos[0].Inicio) = TOD#00:00:00) THEN
           #S_ForaDeTurno := 1;
           #S_TempoRetornoParada := TOD_TO_INT((DTL_TO_TOD(#In_Turnos[0].Inicio))) - TOD_TO_INT(#TOD);
       ELSE
           #S_ForaDeTurno := 0;
           #S_TempoRetornoParada := 0;
       END_IF;

   ELSIF #In_Turnos[1].Fim > #DateTime THEN
       IF NOT (DTL_TO_TOD(#In_Turnos[1].Inicio) = TOD#00:00:00) THEN
           #S_ForaDeTurno := 1;
           #S_TempoRetornoParada := TOD_TO_INT((DTL_TO_TOD(#In_Turnos[1].Inicio))) - TOD_TO_INT(#TOD);
       ELSIF NOT (DTL_TO_TOD(#In_Turnos[2].Inicio) = TOD#00:00:00) THEN
           #S_ForaDeTurno := 1;
           #S_TempoRetornoParada := TOD_TO_INT((DTL_TO_TOD(#In_Turnos[2].Inicio))) - TOD_TO_INT(#TOD);
       ELSIF NOT (DTL_TO_TOD(#In_Turnos[0].Inicio) = TOD#00:00:00) THEN
           #S_ForaDeTurno := 1;
           #S_TempoRetornoParada := TOD_TO_INT((DTL_TO_TOD(#In_Turnos[0].Inicio))) - TOD_TO_INT(#TOD);
       ELSE
           #S_ForaDeTurno := 0;
           #S_TempoRetornoParada := 0;
       END_IF;
   ELSIF #In_Turnos[2].Fim > #DateTime THEN
       IF NOT (DTL_TO_TOD(#In_Turnos[1].Inicio) = TOD#00:00:00) THEN
           #S_ForaDeTurno := 1;
           #S_TempoRetornoParada := TOD_TO_INT((DTL_TO_TOD(#In_Turnos[1].Inicio))) - TOD_TO_INT(#TOD);
       ELSIF NOT (DTL_TO_TOD(#In_Turnos[2].Inicio) = TOD#00:00:00) THEN
           #S_ForaDeTurno := 1;
           #S_TempoRetornoParada := TOD_TO_INT((DTL_TO_TOD(#In_Turnos[2].Inicio))) - TOD_TO_INT(#TOD);
       ELSIF NOT (DTL_TO_TOD(#In_Turnos[0].Inicio) = TOD#00:00:00) THEN
           #S_ForaDeTurno := 1;
           #S_TempoRetornoParada := TOD_TO_INT((DTL_TO_TOD(#In_Turnos[0].Inicio))) - TOD_TO_INT(#TOD);
       ELSE
           #S_ForaDeTurno := 0;
           #S_TempoRetornoParada := 0;
       END_IF;
   END_IF;

   #Out_Parada := #S_ForaDeTurno;
   #Out_TempoRetornoParada := #S_TempoRetornoParada;


   IF #DTL.WEEKDAY = 1 AND "DB303_ScadaToCentral".Data.Dias_Da_Semana[6] THEN
       #Out_EmDiaDeProd :=1;
   ELSIF #DTL.WEEKDAY = 2 AND "DB303_ScadaToCentral".Data.Dias_Da_Semana[0] THEN
       #Out_EmDiaDeProd := 1;
   ELSIF #DTL.WEEKDAY = 3 AND "DB303_ScadaToCentral".Data.Dias_Da_Semana[1] THEN
       #Out_EmDiaDeProd := 1;
   ELSIF #DTL.WEEKDAY = 4 AND "DB303_ScadaToCentral".Data.Dias_Da_Semana[2] THEN
       #Out_EmDiaDeProd := 1;
   ELSIF #DTL.WEEKDAY = 5 AND "DB303_ScadaToCentral".Data.Dias_Da_Semana[3] THEN
       #Out_EmDiaDeProd := 1;
   ELSIF #DTL.WEEKDAY = 6 AND "DB303_ScadaToCentral".Data.Dias_Da_Semana[4] THEN
       #Out_EmDiaDeProd := 1;
   ELSIF #DTL.WEEKDAY = 7 AND "DB303_ScadaToCentral".Data.Dias_Da_Semana[5] THEN
       #Out_EmDiaDeProd := 1;
   ELSE
       #Out_EmDiaDeProd := 0;
   END_IF;
END_FUNCTION_BLOCK

FUNCTION_BLOCK "FB207_ConcatAgvData"   // FB207, SCL
TITLE = FB207_ConcatAgvData
{ S7_Optimized_Access := 'TRUE' }
VERSION : 0.1
// FB207_ConcatAgvData
   VAR_INPUT
      In : Struct   // Dados de entrada do Agv
         Sinais : Byte;
         Posto : Byte;
         Comando : Byte;
         Velocidade : Byte;
         Processo : Byte;
         VelAtual : Byte;
         "Erros.Agv" : Byte;
         "Erros.Pgv" : Byte;
         "Erros.MotorPasso" : Byte;
      END_STRUCT;
      Id : Int;
   END_VAR
   VAR_OUTPUT
      Out : String;   // Saida em formato JSON dos dados do AGV
   END_VAR
   VAR
      Index : Int;
   END_VAR
BEGIN
   (*
       Este bloco realiza a concatenação
       dos dados dos agv e coloca em uma 
       string para que seja possivel enviar 
       o dados em um formato JSON. Caso necessario
       existe a possibilidade de usar-lo quantas
       vezes for necessario.
   *)


   #Out := '';


   #Out := CONCAT(IN1 := '{',
                  IN2 := '"idAgv":"',
                  IN3 := INT_TO_STRING(#Id),
                  IN4 := '","sinais":"',
                  IN5 := INT_TO_STRING(BYTE_TO_INT(#In.Sinais)),
                  IN6 := '","posto":"',
                  IN7 := INT_TO_STRING(BYTE_TO_INT(#In.Posto)),
                  IN8 := '","comando":"',
                  IN9 := INT_TO_STRING(BYTE_TO_INT(#In.Comando)),
                  IN10 := '","velocidade":"',
                  IN11 := INT_TO_STRING(BYTE_TO_INT(#In.Velocidade)),
                  IN12 := '","processo":"',
                  IN13 := INT_TO_STRING(BYTE_TO_INT(#In.Processo)),
                  IN14 := '","velAtual":"',
                  IN15 := INT_TO_STRING(BYTE_TO_INT(#In.VelAtual)),
                  IN16 := '","errosAgv":"',
                  IN17 := INT_TO_STRING(BYTE_TO_INT(#In."Erros.Agv")),
                  IN18 := '","errosPgv":"',
                  IN19 := INT_TO_STRING(BYTE_TO_INT(#In."Erros.Pgv")),
                  IN20 := '","errosMotorPasso":"',
                  IN21 := INT_TO_STRING(BYTE_TO_INT(#In."Erros.MotorPasso")),
                  IN22 := '"}'
   );


       FOR #Index := 0 TO 255 DO
           #Out := CONCAT(IN1 := #Out,
                          IN2 := '-');

       END_FOR;


   (* 
   #Out := CONCAT(IN1 := 'AGV_',
                  IN2 := INT_TO_STRING(#Id),
                  IN3 := ';',
                  IN4 := INT_TO_STRING(BYTE_TO_INT(#In.Sinais)),
                  IN5 := ';',
                  IN6 := INT_TO_STRING(BYTE_TO_INT(#In.Posto)),
                  IN7 := ';',
                  IN8 := INT_TO_STRING(BYTE_TO_INT(#In.Comando)),
                  IN9 := ';',
                  IN10 := INT_TO_STRING(BYTE_TO_INT(#In.Velocidade)),
                  IN11 := ';',
                  IN12 := INT_TO_STRING(BYTE_TO_INT(#In.Processo)),
                  IN13 := ';',
                  IN14 := INT_TO_STRING(BYTE_TO_INT(#In.VelAtual)),
                  IN15 := ';',
                  IN16 := INT_TO_STRING(BYTE_TO_INT(#In."Erros.Agv")),
                  IN17 := ';',
                  IN18 := INT_TO_STRING(BYTE_TO_INT(#In."Erros.Pgv")),
                  IN19 := ';',
                  IN20 := INT_TO_STRING(BYTE_TO_INT(#In."Erros.MotorPasso")),
                  IN21 := '.'
   ); *)
END_FUNCTION_BLOCK

FUNCTION_BLOCK "FB208_ConcatLinhasData"   // FB208, SCL
TITLE = FB208_ConcatLinhasData
{ S7_Optimized_Access := 'TRUE' }
VERSION : 0.1
// FB208_ConcatLinhasData
   VAR_INPUT
      In : Struct   // Dados de entrada da linhas transportadora
         "Timer" : Int;
         StopTime : Int;
         Objetivo : Byte;
         Atual : Byte;
         TempoRetornoParada : Int;
         Andon : Byte;
         Emergencia : Byte;
         CorDeTela : Byte;
         NumMensagem : Byte;
      END_STRUCT;
      Id : String;
   END_VAR
   VAR_OUTPUT
      Out : String;   // Saida em formato JSON dos dados do AGV
   END_VAR
   VAR
      Index : Int;
   END_VAR
BEGIN
   (*
       Este bloco realiza a concatenação
       dos dados das linhas transportadoras e coloca em uma 
       string para que seja possivel enviar 
       o dados em um formato JSON. Caso necessario
       existe a possibilidade de usar-lo quantas
       vezes for necessario.
   *)

   #Out := '';


   #Out := CONCAT(IN1 := '{',
                  IN2 := '"timer":"',
                  IN3 := INT_TO_STRING(#In.Timer),
                  IN4 := '","stopTime":"',
                  IN5 := INT_TO_STRING(#In.StopTime),
                  IN6 := '","objetivo":"',
                  IN7 := INT_TO_STRING(BYTE_TO_INT(#In.Objetivo)),
                  IN8 := '","atual":"',
                  IN9 := INT_TO_STRING(BYTE_TO_INT(#In.Atual)),
                  IN10 := '","tempoRetornoParada":"',
                  IN11 := INT_TO_STRING(#In.TempoRetornoParada),
                  IN12 := '","andon":"',
                  IN13 := INT_TO_STRING(BYTE_TO_INT(#In.Andon)),
                  IN14 := '","emergencia":"',
                  IN15 := INT_TO_STRING(BYTE_TO_INT(#In.Emergencia)),
                  IN16 := '","corDeTela":"',
                  IN17 := INT_TO_STRING(BYTE_TO_INT(#In.CorDeTela)),
                  IN18 := '","numMesagem":"',
                  IN19 := INT_TO_STRING(BYTE_TO_INT(#In.NumMensagem)),
                  IN20 := '","idLine":"',
                  IN21 := #Id,
                  IN22 := '"}'
   );
   FOR #Index := 0 TO 255 DO
       #Out := CONCAT(IN1 := #Out,
                      IN2 := '-');

   END_FOR;
END_FUNCTION_BLOCK

FUNCTION_BLOCK "FB209_FormatadorDados"   // FB209, SCL
TITLE = FB209_FormatadorDados
{ S7_Optimized_Access := 'TRUE' }
VERSION : 0.1
// FB209_FormatadorDados
   VAR_INPUT
      In_Cabinas : Struct
         "Timer" : Int;
         StopTime : Int;
         Objetivo : Byte;
         Atual : Byte;
         TempoRetornoParada : Int;
         Andon : Byte;
         Emergencia : Byte;
         CorDeTela : Byte;
         NumMensagem : Byte;
      END_STRUCT;
      In_Skd : Struct
         "Timer" : Int;
         StopTime : Int;
         Objetivo : Byte;
         Atual : Byte;
         TempoRetornoParada : Int;
         Andon : Byte;
         Emergencia : Byte;
         CorDeTela : Byte;
         NumMensagem : Byte;
      END_STRUCT;
      In_Comp : Struct
         "Timer" : Int;
         StopTime : Int;
         Objetivo : Byte;
         Atual : Byte;
         TempoRetornoParada : Int;
         Andon : Byte;
         Emergencia : Byte;
         CorDeTela : Byte;
         NumMensagem : Byte;
      END_STRUCT;
      In_Ecu : Struct
         "Timer" : Int;
         StopTime : Int;
         Objetivo : Byte;
         Atual : Byte;
         TempoRetornoParada : Int;
         Andon : Byte;
         Emergencia : Byte;
         CorDeTela : Byte;
         NumMensagem : Byte;
      END_STRUCT;
      In_Docas : Array[0..3] of Struct
         "Timer" : Int;
         StopTime : Int;
         Objetivo : Byte;
         Atual : Byte;
         TempoRetornoParada : Int;
         Andon : Byte;
         Emergencia : Byte;
         CorDeTela : Byte;
         NumMensagem : Byte;
      END_STRUCT;
      In_AGVs : Array[0..9] of Struct
         Sinais : Byte;
         Posto : Byte;
         Comando : Byte;
         Velocidade : Byte;
         Processo : Byte;
         VelAtual : Byte;
         "Erros.Agv" : Byte;
         "Erros.Pgv" : Byte;
         "Erros.MotorPasso" : Byte;
      END_STRUCT;
   END_VAR
   VAR_OUTPUT
      Out : Array[0..17] of String;
   END_VAR
   VAR
      ConcatDataAgv : Array[0..9] of "FB207_ConcatAgvData";
      ConcatLinha_Cab : "FB208_ConcatLinhasData";
      ConcatLinha_Skd : "FB208_ConcatLinhasData";
      ConcatLinha_Comp : "FB208_ConcatLinhasData";
      ConcatLinha_Agv : "FB208_ConcatLinhasData";
      ConcatLinha_Doca : Array[0..3] of "FB208_ConcatLinhasData";
      S_DadosAGvs : Array[0..9] of String;
      S_DadosLinhas : Array[0..3] of String;
      S_DadosDocas : Array[0..3] of String;
      S_IndexFor : Int;
      S_IndexFor_2 : Int;
   END_VAR
BEGIN


   REGION FormataDadosDosAgvs
       FOR #S_IndexFor := 0 TO 9 DO
           #ConcatDataAgv[#S_IndexFor](In := #In_AGVs[#S_IndexFor],
                                       Id:=(#S_IndexFor +1) ,
                                       Out => #S_DadosAGvs[#S_IndexFor]);
           #Out[#S_IndexFor] :=  #S_DadosAGvs[#S_IndexFor];
       END_FOR;
   END_REGION


   REGION FormataDadosDasLinhas    
       #ConcatLinha_Cab(In := #In_Cabinas,
                        Id:='CabLine',
                        Out => #S_DadosLinhas[0]);
       #Out[10] := #S_DadosLinhas[0];
       #ConcatLinha_Skd(In := #In_Skd,
                        Id:='SkdLine',
                        Out => #S_DadosLinhas[1]);
       #Out[11] := #S_DadosLinhas[1];
       #ConcatLinha_Comp(In := #In_Comp,
                         Id:='CompLine',
                         Out => #S_DadosLinhas[2]);
       #Out[12] := #S_DadosLinhas[2];
       #ConcatLinha_Agv(In := #In_Ecu,
                        Id:='EcuLine',
                        Out => #S_DadosLinhas[3]);
       #Out[13] := #S_DadosLinhas[3];
   END_REGION

   REGION FormataDadosDasDocas
       FOR #S_IndexFor_2 := 0 TO 3 DO
           #ConcatLinha_Doca[#S_IndexFor_2](In := #In_Docas[#S_IndexFor_2],
                                            Id := CONCAT(IN1 := 'Doca', IN2 := INT_TO_STRING(#S_IndexFor_2 + 1)),
                                            Out => #S_DadosDocas[#S_IndexFor_2]);
       END_FOR;
       #Out[14] := #S_DadosDocas[0];
       #Out[15] := #S_DadosDocas[1];
       #Out[16] := #S_DadosDocas[2];
       #Out[17] := #S_DadosDocas[3];
   END_REGION
END_FUNCTION_BLOCK

FUNCTION_BLOCK "FB212_FomatadorSistemaToPlc"   // FB212, SCL
TITLE = FB212_FomatadorSistemaToPlc
{ S7_Optimized_Access := 'TRUE' }
VERSION : 0.1
// FB212_FomatadorSistemaToPlc
   VAR_INPUT
      "In_Powertrain-Ecu" : "SistemaToTakt";
      In_Componentes : "SistemaToTakt";
      In_Skd : "SistemaToTakt";
      "In_Cabinas-Ecu" : "SistemaToTakt";
      In_Doca1 : "SistemaToTakt";
      In_Doca2 : "SistemaToTakt";
      In_Doca3 : "SistemaToTakt";
      In_Doca4 : "SistemaToTakt";
   END_VAR
   VAR
      FormatadorDadosSistema : "FB213_FormatadorDadosSistema";
      FormatadorDadosSistema_1 : "FB213_FormatadorDadosSistema";
      FormatadorDadosSistema_2 : "FB213_FormatadorDadosSistema";
      FormatadorDadosSistema_3 : "FB213_FormatadorDadosSistema";
      FormatadorDadosSistema_4 : "FB213_FormatadorDadosSistema";
      FormatadorDadosSistema_5 : "FB213_FormatadorDadosSistema";
      FormatadorDadosSistema_6 : "FB213_FormatadorDadosSistema";
      FormatadorDadosSistema_7 : "FB213_FormatadorDadosSistema";
   END_VAR
BEGIN


   REGION Powertrain-Ecu
       #FormatadorDadosSistema(Inicio := #"In_Powertrain-Ecu".Inicio,
                               Fim := #"In_Powertrain-Ecu".Fim,
                               Refeicao := #"In_Powertrain-Ecu".Refeicao,
                               Paradas := #"In_Powertrain-Ecu".Paradas,
                               Out_Inicio=>"DB214_ScadaToLines"."Powertrain-Ecu"[0].Inicio,
                               Out_Fim=>"DB214_ScadaToLines"."Powertrain-Ecu"[0].Fim,
                               Out_RefeicaoInicio=>"DB214_ScadaToLines"."Powertrain-Ecu"[0].RefeicaoInicio,
                               Out_RefeicaoFim=>"DB214_ScadaToLines"."Powertrain-Ecu"[0].RefeicaoFim,
                               Out_Paradas=>"DB214_ScadaToLines"."Powertrain-Ecu"[0].Paradas);
   END_REGION

   REGION Componentes
       #FormatadorDadosSistema_1(Inicio := #"In_Componentes".Inicio,
                                 Fim := #"In_Componentes".Fim,
                                 Refeicao := #"In_Componentes".Refeicao,
                                 Paradas := #"In_Componentes".Paradas,
                                 Out_Inicio=>"DB214_ScadaToLines".Componentes[0].Inicio,
                                 Out_Fim=>"DB214_ScadaToLines".Componentes[0].Fim,
                                 Out_RefeicaoInicio=>"DB214_ScadaToLines".Componentes[0].RefeicaoInicio,
                                 Out_RefeicaoFim=>"DB214_ScadaToLines".Componentes[0].RefeicaoFim,
                                 Out_Paradas=>"DB214_ScadaToLines".Componentes[0].Paradas);
   END_REGION



   REGION Skd
       #FormatadorDadosSistema_2(Inicio := #"In_Skd".Inicio,
                                 Fim := #"In_Skd".Fim,
                                 Refeicao := #"In_Skd".Refeicao,
                                 Paradas := #"In_Skd".Paradas,
                                 Out_Inicio=>"DB214_ScadaToLines".Skd[0].Inicio,
                                 Out_Fim=>"DB214_ScadaToLines".Skd[0].Fim,
                                 Out_RefeicaoInicio=>"DB214_ScadaToLines".Skd[0].RefeicaoInicio,
                                 Out_RefeicaoFim=>"DB214_ScadaToLines".Skd[0].RefeicaoFim,
                                 Out_Paradas=>"DB214_ScadaToLines".Skd[0].Paradas);
   END_REGION

   REGION Cabinas-Ecu
       #FormatadorDadosSistema_3(Inicio := #"In_Cabinas-Ecu".Inicio,
                                 Fim := #"In_Cabinas-Ecu".Fim,
                                 Refeicao := #"In_Cabinas-Ecu".Refeicao,
                                 Paradas := #"In_Cabinas-Ecu".Paradas,
                                 Out_Inicio=>"DB214_ScadaToLines".Cabinas[0].Inicio,
                                 Out_Fim=>"DB214_ScadaToLines".Cabinas[0].Fim,
                                 Out_RefeicaoInicio=>"DB214_ScadaToLines".Cabinas[0].RefeicaoInicio,
                                 Out_RefeicaoFim=>"DB214_ScadaToLines".Cabinas[0].RefeicaoFim,
                                 Out_Paradas=>"DB214_ScadaToLines".Cabinas[0].Paradas);
   END_REGION


   REGION Docas
       REGION Doca 1
           #FormatadorDadosSistema_4(Inicio := #"In_Doca1".Inicio,
                                     Fim := #"In_Doca1".Fim,
                                     Refeicao := #"In_Doca1".Refeicao,
                                     Paradas := #"In_Doca1".Paradas);
       END_REGION
       REGION Doca 2        
           #FormatadorDadosSistema_5(Inicio := #"In_Doca2".Inicio,
                                     Fim := #"In_Doca2".Fim,
                                     Refeicao := #"In_Doca2".Refeicao,
                                     Paradas := #"In_Doca2".Paradas);
       END_REGION
       REGION Doca 3        
           #FormatadorDadosSistema_6(Inicio := #"In_Doca3".Inicio,
                                     Fim := #"In_Doca3".Fim,
                                     Refeicao := #"In_Doca3".Refeicao,
                                     Paradas := #"In_Doca3".Paradas);
       END_REGION
       REGION Doca 4
           #FormatadorDadosSistema_7(Inicio := #"In_Doca4".Inicio,
                                     Fim := #"In_Doca4".Fim,
                                     Refeicao := #"In_Doca4".Refeicao,
                                     Paradas := #"In_Doca4".Paradas);
       END_REGION

   END_REGION
END_FUNCTION_BLOCK

FUNCTION_BLOCK "FB213_FormatadorDadosSistema"   // FB213, SCL
TITLE = FB213_FormatadorDadosSistema
{ S7_Optimized_Access := 'TRUE' }
VERSION : 0.1
// FB213_FormatadorDadosSistema
   VAR_INPUT
      Inicio : Array[0..4] of Int;
      Fim : Array[0..4] of Int;
      Refeicao : Array[0..4] of Int;
      Paradas : Array[0..4] of Struct
         Inicio : Array[0..4] of Int;
         Fim : Array[0..4] of Int;
      END_STRUCT;
   END_VAR
   VAR_OUTPUT
      Out_Inicio : DTL;
      Out_Fim : DTL;
      Out_RefeicaoInicio : DTL;
      Out_RefeicaoFim : DTL;
      Out_Paradas : Array[0..4] of Struct
         Inicio : DTL;
         Fim : DTL;
      END_STRUCT;
      Index : Int;
   END_VAR
   // // Inicio[0] : Ano
   // // Inicio[1] : Mês
   // // Inicio[2] : Dia
   // // Inicio[3] : Hora
   // // Inicio[4] : Minuto
   // // Fim[0] : Ano
   // // Fim[1] : Mês
   // // Fim[2] : Dia
   // // Fim[3] : Hora
   // // Fim[4] : Minuto
   // // Refeicao[0] : Ano
   // // Refeicao[1] : Mês
   // // Refeicao[2] : Dia
   // // Refeicao[3] : Hora
   // // Refeicao[4] : Minuto
   // // Paradas[0].Inicio[0] : Ano
   // // Paradas[0].Inicio[1] : Mês
   // // Paradas[0].Inicio[2] : Dia
   // // Paradas[0].Inicio[3] : Hora
   // // Paradas[0].Inicio[4] : Minuto
   // // Paradas[0].Fim[0] : Ano
   // // Paradas[0].Fim[1] : Mês
   // // Paradas[0].Fim[2] : Dia
   // // Paradas[0].Fim[3] : Hora
   // // Paradas[0].Fim[4] : Minuto
BEGIN







   REGION ConversorInicioTurno
       #Out_Inicio.YEAR := INT_TO_UINT(#Inicio[0]);
       #Out_Inicio.MONTH := INT_TO_USINT(#Inicio[1]);
       #Out_Inicio.DAY := INT_TO_USINT(#Inicio[2]);
       #Out_Inicio.HOUR := INT_TO_USINT(#Inicio[3]);
       #Out_Inicio.MINUTE := INT_TO_USINT(#Inicio[4]);
       #Out_Inicio.SECOND := 00;

   END_REGION


   REGION ConversorFimTurno
       #Out_Fim.YEAR :=  INT_TO_UINT(#Fim[0]);
       #Out_Fim.MONTH := INT_TO_USINT(#Fim[1]);
       #Out_Fim.DAY :=   INT_TO_USINT(#Fim[2]);
       #Out_Fim.HOUR :=  INT_TO_USINT(#Fim[3]);
       #Out_Fim.MINUTE :=INT_TO_USINT(#Fim[4]);
       #Out_Fim.SECOND := 00;

   END_REGION


   REGION ConversorRefeicaoInicio
       #Out_Fim.YEAR := INT_TO_UINT(#Fim[0]);
       #Out_Fim.MONTH := INT_TO_USINT(#Fim[1]);
       #Out_Fim.DAY := INT_TO_USINT(#Fim[2]);
       #Out_Fim.HOUR := INT_TO_USINT(#Fim[3]);
       #Out_Fim.MINUTE := INT_TO_USINT(#Fim[4]);
       #Out_Fim.SECOND := 00;

   END_REGION


   REGION ConversorRefeicaoInicio
       #Out_RefeicaoInicio.YEAR := INT_TO_UINT(#Refeicao[0]);
       #Out_RefeicaoInicio.MONTH := INT_TO_USINT(#Refeicao[1]);
       #Out_RefeicaoInicio.DAY := INT_TO_USINT(#Refeicao[2]);
       #Out_RefeicaoInicio.HOUR := INT_TO_USINT(#Refeicao[3]);
       #Out_RefeicaoInicio.MINUTE := INT_TO_USINT(#Refeicao[4]);
       #Out_RefeicaoInicio.SECOND := 00;

   END_REGION

   REGION ConversorRefeicaoFim
       #Out_RefeicaoFim.YEAR := INT_TO_UINT(#Refeicao[0]);
       #Out_RefeicaoFim.MONTH := INT_TO_USINT(#Refeicao[1]);
       #Out_RefeicaoFim.DAY := INT_TO_USINT(#Refeicao[2]);
       #Out_RefeicaoFim.HOUR := INT_TO_USINT(#Refeicao[3]+1);
       #Out_RefeicaoFim.MINUTE := INT_TO_USINT(#Refeicao[4]);
       #Out_RefeicaoFim.SECOND := 00;

   END_REGION


   FOR #Index := 0 TO 4 DO
       IF #Paradas[#Index].Inicio[0] = 0 OR #Paradas[#Index].Inicio[1] = 0 OR #Paradas[#Index].Inicio[2] = 0THEN

           #Out_Paradas[#Index].Inicio.YEAR := 1970;
           #Out_Paradas[#Index].Inicio.MONTH := 01;
           #Out_Paradas[#Index].Inicio.DAY := 01;
           #Out_Paradas[#Index].Inicio.HOUR := 00;
           #Out_Paradas[#Index].Inicio.MINUTE := 00;
           #Out_Paradas[#Index].Inicio.SECOND := 00;

           #Out_Paradas[#Index].Fim.YEAR := 1970;
           #Out_Paradas[#Index].Fim.MONTH := 01;
           #Out_Paradas[#Index].Fim.DAY := 01;
           #Out_Paradas[#Index].Fim.HOUR := 0;
           #Out_Paradas[#Index].Fim.MINUTE := 00;
           #Out_Paradas[#Index].Fim.SECOND := 00;
       ELSE
           #Out_Paradas[#Index].Inicio.YEAR := INT_TO_UINT(#Paradas[#Index].Inicio[0]);
           #Out_Paradas[#Index].Inicio.MONTH := INT_TO_USINT(#Paradas[#Index].Inicio[1]);
           #Out_Paradas[#Index].Inicio.DAY := INT_TO_USINT(#Paradas[#Index].Inicio[2]);
           #Out_Paradas[#Index].Inicio.HOUR := INT_TO_USINT(#Paradas[#Index].Inicio[3]);
           #Out_Paradas[#Index].Inicio.MINUTE := INT_TO_USINT(#Paradas[#Index].Inicio[4]);
           #Out_Paradas[#Index].Inicio.SECOND := 00;

           #Out_Paradas[#Index].Fim.YEAR := INT_TO_UINT(#Paradas[#Index].Fim[0]);
           #Out_Paradas[#Index].Fim.MONTH := INT_TO_USINT(#Paradas[#Index].Fim[1]);
           #Out_Paradas[#Index].Fim.DAY := INT_TO_USINT(#Paradas[#Index].Fim[2]);
           #Out_Paradas[#Index].Fim.HOUR := INT_TO_USINT(#Paradas[#Index].Fim[3]);
           #Out_Paradas[#Index].Fim.MINUTE := INT_TO_USINT(#Paradas[#Index].Fim[4]);
           #Out_Paradas[#Index].Fim.SECOND := 00;
       END_IF;



   END_FOR;
END_FUNCTION_BLOCK

// folder: 04_Services/01_FB

FUNCTION_BLOCK "FB400_Clock_Regulavel"   // FB400, SCL
{ S7_Optimized_Access := 'TRUE' }
VERSION : 0.1
   VAR_INPUT
      In_Tempo : Time;
   END_VAR
   VAR_OUTPUT
      Out_Pulso : Bool;
      Out_Sinal : Bool;
      Out_NotSinal : Bool;
   END_VAR
   VAR
      TON_1 : TON_TIME;
      TON_2 : TON_TIME;
      R_TRIG_Instance : R_TRIG;
   END_VAR
BEGIN


   #TON_1(IN:= NOT #TON_2.Q,
          PT:=#In_Tempo);


   #TON_2(IN := #TON_1.Q,
          PT := #In_Tempo);

   #R_TRIG_Instance(CLK:=#Out_Sinal);


   #Out_Sinal := #TON_1.Q;
   #Out_NotSinal := NOT #TON_1.Q;
   #Out_Pulso := #R_TRIG_Instance.Q;
END_FUNCTION_BLOCK

(* ===== HMI "HMI_RT_1" =====
system functions are stored by id; their names below are inferred from use
connection "HMI_CENTRAL": ETHERNET, S7_1500_OMS

HMI tags "Default tag table"
   "DB300_IhmDados_Dados_Cabinas_Tempo_Takt" : DInt = PLC DB300_IhmDados.Dados_Cabinas.Tempo_Takt AT %DB300.DBD0, 1 s
   "DB300_IhmDados_Dados_Cabinas_Tempo_StopTime" : DInt = PLC DB300_IhmDados.Dados_Cabinas.Tempo_StopTime AT %DB300.DBD4, 1 s
   "DB300_IhmDados_Dados_Cabinas_Objetivo" : Int = PLC DB300_IhmDados.Dados_Cabinas.Objetivo AT %DB300.DBW8, 1 s
   "DB300_IhmDados_Dados_Cabinas_Atual" : Int = PLC DB300_IhmDados.Dados_Cabinas.Atual AT %DB300.DBW10, 1 s
   "DB300_IhmDados_Dados_Cabinas_DirectRun" : Real = PLC DB300_IhmDados.Dados_Cabinas.DirectRun AT %DB300.DBD24, 1 s
   "DB300_IhmDados_Dados_Cabinas_SaldoDoTurno" : Int = PLC DB300_IhmDados.Dados_Cabinas.SaldoDoTurno AT %DB300.DBW28, 1 s
   "DB300_IhmDados_Dados_Cabinas_Andons{0}" : Bool = PLC DB300_IhmDados.Dados_Cabinas.Andons[0] AT %DB300.DBX20.0, 1 s
   "DB300_IhmDados_Dados_Cabinas_Andons{1}" : Bool = PLC DB300_IhmDados.Dados_Cabinas.Andons[1] AT %DB300.DBX20.1, 1 s
   "DB300_IhmDados_Dados_Cabinas_Andons{2}" : Bool = PLC DB300_IhmDados.Dados_Cabinas.Andons[2] AT %DB300.DBX20.2, 1 s
   "DB300_IhmDados_Dados_Cabinas_Andons{3}" : Bool = PLC DB300_IhmDados.Dados_Cabinas.Andons[3] AT %DB300.DBX20.3, 1 s
   "DB300_IhmDados_Dados_Cabinas_Andons{4}" : Bool = PLC DB300_IhmDados.Dados_Cabinas.Andons[4] AT %DB300.DBX20.4, 1 s
   "DB300_IhmDados_Dados_Cabinas_Andons{5}" : Bool = PLC DB300_IhmDados.Dados_Cabinas.Andons[5] AT %DB300.DBX20.5, 1 s
   "DB300_IhmDados_Dados_Cabinas_Andons{6}" : Bool = PLC DB300_IhmDados.Dados_Cabinas.Andons[6] AT %DB300.DBX20.6, 1 s
   "DB300_IhmDados_Dados_Cabinas_Andons{7}" : Bool = PLC DB300_IhmDados.Dados_Cabinas.Andons[7] AT %DB300.DBX20.7, 1 s
   "DB300_IhmDados_Dados_Cabinas_CorDeTela" : Byte = PLC DB300_IhmDados.Dados_Cabinas.CorDeTela AT %DB300.DBB22, 1 s
   "DB300_IhmDados_Mensagem_Cab" : String[254] = PLC DB300_IhmDados.Mensagem_Cab AT %DB300.DBX64.0, 1 s
   "DB300_IhmDados_Dados_ECU_Andons{0}" : Bool = PLC DB300_IhmDados.Dados_ECU.Andons[0] AT %DB300.DBX980.0, 1 s
   "DB300_IhmDados_Dados_ECU_Andons{1}" : Bool = PLC DB300_IhmDados.Dados_ECU.Andons[1] AT %DB300.DBX980.1, 1 s
   "DB300_IhmDados_Dados_ECU_Andons{2}" : Bool = PLC DB300_IhmDados.Dados_ECU.Andons[2] AT %DB300.DBX980.2, 1 s
   "DB300_IhmDados_Dados_ECU_Andons{3}" : Bool = PLC DB300_IhmDados.Dados_ECU.Andons[3] AT %DB300.DBX980.3, 1 s
   "DB300_IhmDados_Dados_ECU_Andons{4}" : Bool = PLC DB300_IhmDados.Dados_ECU.Andons[4] AT %DB300.DBX980.4, 1 s
   "DB300_IhmDados_Dados_ECU_Andons{5}" : Bool = PLC DB300_IhmDados.Dados_ECU.Andons[5] AT %DB300.DBX980.5, 1 s
   "DB300_IhmDados_Dados_ECU_Andons{6}" : Bool = PLC DB300_IhmDados.Dados_ECU.Andons[6] AT %DB300.DBX980.6, 1 s
   "DB300_IhmDados_Dados_ECU_Andons{7}" : Bool = PLC DB300_IhmDados.Dados_ECU.Andons[7] AT %DB300.DBX980.7, 1 s
   "DB300_IhmDados_Dados_ECU_Tempo_StopTime" : DInt = PLC DB300_IhmDados.Dados_ECU.Tempo_StopTime AT %DB300.DBD964, 1 s
   "DB300_IhmDados_Dados_ECU_Tempo_Takt" : DInt = PLC DB300_IhmDados.Dados_ECU.Tempo_Takt AT %DB300.DBD960, 1 s
   "DB300_IhmDados_Dados_ECU_Objetivo" : Int = PLC DB300_IhmDados.Dados_ECU.Objetivo AT %DB300.DBW968, 1 s
   "DB300_IhmDados_Dados_ECU_Atual" : Int = PLC DB300_IhmDados.Dados_ECU.Atual AT %DB300.DBW970, 1 s
   "DB300_IhmDados_Dados_ECU_DirectRun" : Real = PLC DB300_IhmDados.Dados_ECU.DirectRun AT %DB300.DBD984, 1 s
   "DB300_IhmDados_Dados_ECU_SaldoDoTurno" : Int = PLC DB300_IhmDados.Dados_ECU.SaldoDoTurno AT %DB300.DBW988, 1 s
   "DB300_IhmDados_Mensagem_ECU" : String[254] = PLC DB300_IhmDados.Mensagem_ECU AT %DB300.DBX1024.0, 1 s
   "DB300_IhmDados_Dados_ECU_CorDeTela" : Byte = PLC DB300_IhmDados.Dados_ECU.CorDeTela AT %DB300.DBB982, 1 s
   "DB300_IhmDados_Dados_SKD_Tempo_Takt" : DInt = PLC DB300_IhmDados.Dados_SKD.Tempo_Takt AT %DB300.DBD320, 1 s
   "DB300_IhmDados_Dados_SKD_Tempo_StopTime" : DInt = PLC DB300_IhmDados.Dados_SKD.Tempo_StopTime AT %DB300.DBD324, 1 s
   "DB300_IhmDados_Dados_SKD_Objetivo" : Int = PLC DB300_IhmDados.Dados_SKD.Objetivo AT %DB300.DBW328, 1 s
   "DB300_IhmDados_Dados_SKD_Atual" : Int = PLC DB300_IhmDados.Dados_SKD.Atual AT %DB300.DBW330, 1 s
   "DB300_IhmDados_Dados_SKD_DirectRun" : Real = PLC DB300_IhmDados.Dados_SKD.DirectRun AT %DB300.DBD344, 1 s
   "DB300_IhmDados_Dados_SKD_SaldoDoTurno" : Int = PLC DB300_IhmDados.Dados_SKD.SaldoDoTurno AT %DB300.DBW348, 1 s
   "DB300_IhmDados_Mensagem_SKD" : String[254] = PLC DB300_IhmDados.Mensagem_SKD AT %DB300.DBX384.0, 1 s
   "DB300_IhmDados_Dados_SKD_CorDeTela" : Byte = PLC DB300_IhmDados.Dados_SKD.CorDeTela AT %DB300.DBB342, 1 s
   "DB300_IhmDados_Dados_SKD_Andons{0}" : Bool = PLC DB300_IhmDados.Dados_SKD.Andons[0] AT %DB300.DBX340.0, 1 s
   "DB300_IhmDados_Dados_SKD_Andons{1}" : Bool = PLC DB300_IhmDados.Dados_SKD.Andons[1] AT %DB300.DBX340.1, 1 s
   "DB300_IhmDados_Dados_SKD_Andons{2}" : Bool = PLC DB300_IhmDados.Dados_SKD.Andons[2] AT %DB300.DBX340.2, 1 s
   "DB300_IhmDados_Dados_SKD_Andons{3}" : Bool = PLC DB300_IhmDados.Dados_SKD.Andons[3] AT %DB300.DBX340.3, 1 s
   "DB300_IhmDados_Dados_SKD_Andons{4}" : Bool = PLC DB300_IhmDados.Dados_SKD.Andons[4] AT %DB300.DBX340.4, 1 s
   "DB300_IhmDados_Dados_SKD_Andons{5}" : Bool = PLC DB300_IhmDados.Dados_SKD.Andons[5] AT %DB300.DBX340.5, 1 s
   "DB300_IhmDados_Dados_SKD_Andons{6}" : Bool = PLC DB300_IhmDados.Dados_SKD.Andons[6] AT %DB300.DBX340.6, 1 s
   "DB300_IhmDados_Dados_SKD_Andons{7}" : Bool = PLC DB300_IhmDados.Dados_SKD.Andons[7] AT %DB300.DBX340.7, 1 s
   "DB300_IhmDados_Dados_Componentes_Andons{0}" : Bool = PLC DB300_IhmDados.Dados_Componentes.Andons[0] AT %DB300.DBX660.0, 1 s
   "DB300_IhmDados_Dados_Componentes_Andons{1}" : Bool = PLC DB300_IhmDados.Dados_Componentes.Andons[1] AT %DB300.DBX660.1, 1 s
   "DB300_IhmDados_Dados_Componentes_Andons{2}" : Bool = PLC DB300_IhmDados.Dados_Componentes.Andons[2] AT %DB300.DBX660.2, 1 s
   "DB300_IhmDados_Dados_Componentes_Andons{3}" : Bool = PLC DB300_IhmDados.Dados_Componentes.Andons[3] AT %DB300.DBX660.3, 1 s
   "DB300_IhmDados_Dados_Componentes_Andons{4}" : Bool = PLC DB300_IhmDados.Dados_Componentes.Andons[4] AT %DB300.DBX660.4, 1 s
   "DB300_IhmDados_Dados_Componentes_Andons{5}" : Bool = PLC DB300_IhmDados.Dados_Componentes.Andons[5] AT %DB300.DBX660.5, 1 s
   "DB300_IhmDados_Dados_Componentes_Andons{6}" : Bool = PLC DB300_IhmDados.Dados_Componentes.Andons[6] AT %DB300.DBX660.6, 1 s
   "DB300_IhmDados_Dados_Componentes_Andons{7}" : Bool = PLC DB300_IhmDados.Dados_Componentes.Andons[7] AT %DB300.DBX660.7, 1 s
   "DB300_IhmDados_Dados_Componentes_Tempo_Takt" : DInt = PLC DB300_IhmDados.Dados_Componentes.Tempo_Takt AT %DB300.DBD640, 1 s
   "DB300_IhmDados_Dados_Componentes_Tempo_StopTime" : DInt = PLC DB300_IhmDados.Dados_Componentes.Tempo_StopTime AT %DB300.DBD644, 1 s
   "DB300_IhmDados_Dados_Componentes_Objetivo" : Int = PLC DB300_IhmDados.Dados_Componentes.Objetivo AT %DB300.DBW648, 1 s
   "DB300_IhmDados_Dados_Componentes_Atual" : Int = PLC DB300_IhmDados.Dados_Componentes.Atual AT %DB300.DBW650, 1 s
   "DB300_IhmDados_Dados_Componentes_DirectRun" : Real = PLC DB300_IhmDados.Dados_Componentes.DirectRun AT %DB300.DBD664, 1 s
   "DB300_IhmDados_Dados_Componentes_SaldoDoTurno" : Int = PLC DB300_IhmDados.Dados_Componentes.SaldoDoTurno AT %DB300.DBW668, 1 s
   "DB300_IhmDados_Mensagem_Componentes" : String[254] = PLC DB300_IhmDados.Mensagem_Componentes AT %DB300.DBX704.0, 1 s
   "DB300_IhmDados_Dados_Componentes_CorDeTela" : Byte = PLC DB300_IhmDados.Dados_Componentes.CorDeTela AT %DB300.DBB662, 1 s
   "DB302_InputDados_Ecu_SistemaOn" : Bool = PLC DB302_InputDados.Ecu.SistemaOn AT %DB302.DBX180.0, 1 s
   "DB302_InputDados_Ecu_Turnos_1_Turno_Inicio" : Date_And_Time = PLC DB302_InputDados.Ecu.Turnos.1_Turno.Inicio AT %DB302.DBX0.0, 1 s
   "DB302_InputDados_Ecu_Turnos_1_Turno_Fim" : Date_And_Time = PLC DB302_InputDados.Ecu.Turnos.1_Turno.Fim AT %DB302.DBX8.0, 1 s
   "DB302_InputDados_Ecu_Turnos_1_Turno_TempoTakt" : Int = PLC DB302_InputDados.Ecu.Turnos.1_Turno.TempoTakt AT %DB302.DBW16, 1 s
   "DB302_InputDados_Ecu_Turnos_1_Turno_Rodadas" : Int = PLC DB302_InputDados.Ecu.Turnos.1_Turno.Rodadas AT %DB302.DBW18, 1 s
   "DB302_InputDados_Ecu_Turnos_2_Turno_Inicio" : Date_And_Time = PLC DB302_InputDados.Ecu.Turnos.2_Turno.Inicio AT %DB302.DBX20.0, 1 s
   "DB302_InputDados_Ecu_Turnos_2_Turno_Fim" : Date_And_Time = PLC DB302_InputDados.Ecu.Turnos.2_Turno.Fim AT %DB302.DBX28.0, 1 s
   "DB302_InputDados_Ecu_Turnos_2_Turno_TempoTakt" : Int = PLC DB302_InputDados.Ecu.Turnos.2_Turno.TempoTakt AT %DB302.DBW36, 1 s
   "DB302_InputDados_Ecu_Turnos_2_Turno_Rodadas" : Int = PLC DB302_InputDados.Ecu.Turnos.2_Turno.Rodadas AT %DB302.DBW38, 1 s
   "DB302_InputDados_Ecu_Turnos_3_Turno_TempoTakt" : Int = PLC DB302_InputDados.Ecu.Turnos.3_Turno.TempoTakt AT %DB302.DBW56, 1 s
   "DB302_InputDados_Ecu_Turnos_3_Turno_Rodadas" : Int = PLC DB302_InputDados.Ecu.Turnos.3_Turno.Rodadas AT %DB302.DBW58, 1 s
   "DB302_InputDados_Ecu_Turnos_3_Turno_Fim" : Date_And_Time = PLC DB302_InputDados.Ecu.Turnos.3_Turno.Fim AT %DB302.DBX48.0, 1 s
   "DB302_InputDados_Ecu_Turnos_3_Turno_Inicio" : Date_And_Time = PLC DB302_InputDados.Ecu.Turnos.3_Turno.Inicio AT %DB302.DBX40.0, 1 s
   "DB302_InputDados_Ecu_Paradas_Programadas_1Turno_Parada_1_Inicio" : Time_Of_Day = PLC DB302_InputDados.Ecu.Paradas_Programadas_1Turno.Parada_1.Inicio AT %DB302.DBD60, 1 s
   "DB302_InputDados_Ecu_Paradas_Programadas_1Turno_Parada_1_Fim" : Time_Of_Day = PLC DB302_InputDados.Ecu.Paradas_Programadas_1Turno.Parada_1.Fim AT %DB302.DBD64, 1 s
   "DB302_InputDados_Ecu_Paradas_Programadas_1Turno_Parada_2_Inicio" : Time_Of_Day = PLC DB302_InputDados.Ecu.Paradas_Programadas_1Turno.Parada_2.Inicio AT %DB302.DBD68, 1 s
   "DB302_InputDados_Ecu_Paradas_Programadas_1Turno_Parada_2_Fim" : Time_Of_Day = PLC DB302_InputDados.Ecu.Paradas_Programadas_1Turno.Parada_2.Fim AT %DB302.DBD72, 1 s
   "DB302_InputDados_Ecu_Paradas_Programadas_1Turno_Parada_3_Inicio" : Time_Of_Day = PLC DB302_InputDados.Ecu.Paradas_Programadas_1Turno.Parada_3.Inicio AT %DB302.DBD76, 1 s
   "DB302_InputDados_Ecu_Paradas_Programadas_1Turno_Parada_3_Fim" : Time_Of_Day = PLC DB302_InputDados.Ecu.Paradas_Programadas_1Turno.Parada_3.Fim AT %DB302.DBD80, 1 s
   "DB302_InputDados_Ecu_Paradas_Programadas_1Turno_Parada_4_Inicio" : Time_Of_Day = PLC DB302_InputDados.Ecu.Paradas_Programadas_1Turno.Parada_4.Inicio AT %DB302.DBD84, 1 s
   "DB302_InputDados_Ecu_Paradas_Programadas_1Turno_Parada_4_Fim" : Time_Of_Day = PLC DB302_InputDados.Ecu.Paradas_Programadas_1Turno.Parada_4.Fim AT %DB302.DBD88, 1 s
   "DB302_InputDados_Ecu_Paradas_Programadas_1Turno_Parada_5_Inicio" : Time_Of_Day = PLC DB302_InputDados.Ecu.Paradas_Programadas_1Turno.Parada_5.Inicio AT %DB302.DBD92, 1 s
   "DB302_InputDados_Ecu_Paradas_Programadas_1Turno_Parada_5_Fim" : Time_Of_Day = PLC DB302_InputDados.Ecu.Paradas_Programadas_1Turno.Parada_5.Fim AT %DB302.DBD96, 1 s
   "DB302_InputDados_Ecu_Paradas_Programadas_2Turno_Parada_1_Inicio" : Time_Of_Day = PLC DB302_InputDados.Ecu.Paradas_Programadas_2Turno.Parada_1.Inicio AT %DB302.DBD100, 1 s
   "DB302_InputDados_Ecu_Paradas_Programadas_2Turno_Parada_1_Fim" : Time_Of_Day = PLC DB302_InputDados.Ecu.Paradas_Programadas_2Turno.Parada_1.Fim AT %DB302.DBD104, 1 s
   "DB302_InputDados_Ecu_Paradas_Programadas_2Turno_Parada_2_Inicio" : Time_Of_Day = PLC DB302_InputDados.Ecu.Paradas_Programadas_2Turno.Parada_2.Inicio AT %DB302.DBD108, 1 s
   "DB302_InputDados_Ecu_Paradas_Programadas_2Turno_Parada_2_Fim" : Time_Of_Day = PLC DB302_InputDados.Ecu.Paradas_Programadas_2Turno.Parada_2.Fim AT %DB302.DBD112, 1 s
   "DB302_InputDados_Ecu_Paradas_Programadas_2Turno_Parada_3_Inicio" : Time_Of_Day = PLC DB302_InputDados.Ecu.Paradas_Programadas_2Turno.Parada_3.Inicio AT %DB302.DBD116, 1 s
   "DB302_InputDados_Ecu_Paradas_Programadas_2Turno_Parada_3_Fim" : Time_Of_Day = PLC DB302_InputDados.Ecu.Paradas_Programadas_2Turno.Parada_3.Fim AT %DB302.DBD120, 1 s
   "DB302_InputDados_Ecu_Paradas_Programadas_2Turno_Parada_4_Inicio" : Time_Of_Day = PLC DB302_InputDados.Ecu.Paradas_Programadas_2Turno.Parada_4.Inicio AT %DB302.DBD124, 1 s
   "DB302_InputDados_Ecu_Paradas_Programadas_2Turno_Parada_4_Fim" : Time_Of_Day = PLC DB302_InputDados.Ecu.Paradas_Programadas_2Turno.Parada_4.Fim AT %DB302.DBD128, 1 s
   "DB302_InputDados_Ecu_Paradas_Programadas_2Turno_Parada_5_Inicio" : Time_Of_Day = PLC DB302_InputDados.Ecu.Paradas_Programadas_2Turno.Parada_5.Inicio AT %DB302.DBD132, 1 s
   "DB302_InputDados_Ecu_Paradas_Programadas_2Turno_Parada_5_Fim" : Time_Of_Day = PLC DB302_InputDados.Ecu.Paradas_Programadas_2Turno.Parada_5.Fim AT %DB302.DBD136, 1 s
   "DB302_InputDados_Ecu_Paradas_Programadas_3Turno_Parada_1_Inicio" : Time_Of_Day = PLC DB302_InputDados.Ecu.Paradas_Programadas_3Turno.Parada_1.Inicio AT %DB302.DBD140, 1 s
   "DB302_InputDados_Ecu_Paradas_Programadas_3Turno_Parada_1_Fim" : Time_Of_Day = PLC DB302_InputDados.Ecu.Paradas_Programadas_3Turno.Parada_1.Fim AT %DB302.DBD144, 1 s
   "DB302_InputDados_Ecu_Paradas_Programadas_3Turno_Parada_2_Inicio" : Time_Of_Day = PLC DB302_InputDados.Ecu.Paradas_Programadas_3Turno.Parada_2.Inicio AT %DB302.DBD148, 1 s
   "DB302_InputDados_Ecu_Paradas_Programadas_3Turno_Parada_2_Fim" : Time_Of_Day = PLC DB302_InputDados.Ecu.Paradas_Programadas_3Turno.Parada_2.Fim AT %DB302.DBD152, 1 s
   "DB302_InputDados_Ecu_Paradas_Programadas_3Turno_Parada_3_Inicio" : Time_Of_Day = PLC DB302_InputDados.Ecu.Paradas_Programadas_3Turno.Parada_3.Inicio AT %DB302.DBD156, 1 s
   "DB302_InputDados_Ecu_Paradas_Programadas_3Turno_Parada_3_Fim" : Time_Of_Day = PLC DB302_InputDados.Ecu.Paradas_Programadas_3Turno.Parada_3.Fim AT %DB302.DBD160, 1 s
   "DB302_InputDados_Ecu_Paradas_Programadas_3Turno_Parada_4_Inicio" : Time_Of_Day = PLC DB302_InputDados.Ecu.Paradas_Programadas_3Turno.Parada_4.Inicio AT %DB302.DBD164, 1 s
   "DB302_InputDados_Ecu_Paradas_Programadas_3Turno_Parada_4_Fim" : Time_Of_Day = PLC DB302_InputDados.Ecu.Paradas_Programadas_3Turno.Parada_4.Fim AT %DB302.DBD168, 1 s
   "DB302_InputDados_Ecu_Paradas_Programadas_3Turno_Parada_5_Inicio" : Time_Of_Day = PLC DB302_InputDados.Ecu.Paradas_Programadas_3Turno.Parada_5.Inicio AT %DB302.DBD172, 1 s
   "DB302_InputDados_Ecu_Paradas_Programadas_3Turno_Parada_5_Fim" : Time_Of_Day = PLC DB302_InputDados.Ecu.Paradas_Programadas_3Turno.Parada_5.Fim AT %DB302.DBD176, 1 s
   "DB302_InputDados_Cabinas_Turnos_1_Turno_Inicio" : Date_And_Time = PLC DB302_InputDados.Cabinas.Turnos.1_Turno.Inicio AT %DB302.DBX182.0, 1 s
   "DB302_InputDados_Cabinas_Turnos_1_Turno_Fim" : Date_And_Time = PLC DB302_InputDados.Cabinas.Turnos.1_Turno.Fim AT %DB302.DBX190.0, 1 s
   "DB302_InputDados_Cabinas_Turnos_1_Turno_TempoTakt" : Int = PLC DB302_InputDados.Cabinas.Turnos.1_Turno.TempoTakt AT %DB302.DBW198, 1 s
   "DB302_InputDados_Cabinas_Turnos_1_Turno_Rodadas" : Int = PLC DB302_InputDados.Cabinas.Turnos.1_Turno.Rodadas AT %DB302.DBW200, 1 s
   "DB302_InputDados_Cabinas_Turnos_2_Turno_Inicio" : Date_And_Time = PLC DB302_InputDados.Cabinas.Turnos.2_Turno.Inicio AT %DB302.DBX202.0, 1 s
   "DB302_InputDados_Cabinas_Turnos_2_Turno_Fim" : Date_And_Time = PLC DB302_InputDados.Cabinas.Turnos.2_Turno.Fim AT %DB302.DBX210.0, 1 s
   "DB302_InputDados_Cabinas_Turnos_2_Turno_TempoTakt" : Int = PLC DB302_InputDados.Cabinas.Turnos.2_Turno.TempoTakt AT %DB302.DBW218, 1 s
   "DB302_InputDados_Cabinas_Turnos_2_Turno_Rodadas" : Int = PLC DB302_InputDados.Cabinas.Turnos.2_Turno.Rodadas AT %DB302.DBW220, 1 s
   "DB302_InputDados_Cabinas_Turnos_3_Turno_Inicio" : Date_And_Time = PLC DB302_InputDados.Cabinas.Turnos.3_Turno.Inicio AT %DB302.DBX222.0, 1 s
   "DB302_InputDados_Cabinas_Turnos_3_Turno_Fim" : Date_And_Time = PLC DB302_InputDados.Cabinas.Turnos.3_Turno.Fim AT %DB302.DBX230.0, 1 s
   "DB302_InputDados_Cabinas_Turnos_3_Turno_TempoTakt" : Int = PLC DB302_InputDados.Cabinas.Turnos.3_Turno.TempoTakt AT %DB302.DBW238, 1 s
   "DB302_InputDados_Cabinas_Turnos_3_Turno_Rodadas" : Int = PLC DB302_InputDados.Cabinas.Turnos.3_Turno.Rodadas AT %DB302.DBW240, 1 s
   "DB302_InputDados_Cabinas_SistemaOn" : Bool = PLC DB302_InputDados.Cabinas.SistemaOn AT %DB302.DBX362.0, 1 s
   "DB302_InputDados_SKD_Turnos_1_Turno_Inicio" : Date_And_Time = PLC DB302_InputDados.SKD.Turnos.1_Turno.Inicio AT %DB302.DBX364.0, 1 s
   "DB302_InputDados_SKD_Turnos_1_Turno_Fim" : Date_And_Time = PLC DB302_InputDados.SKD.Turnos.1_Turno.Fim AT %DB302.DBX372.0, 1 s
   "DB302_InputDados_SKD_Turnos_1_Turno_TempoTakt" : Int = PLC DB302_InputDados.SKD.Turnos.1_Turno.TempoTakt AT %DB302.DBW380, 1 s
   "DB302_InputDados_SKD_Turnos_1_Turno_Rodadas" : Int = PLC DB302_InputDados.SKD.Turnos.1_Turno.Rodadas AT %DB302.DBW382, 1 s
   "DB302_InputDados_SKD_Turnos_2_Turno_Inicio" : Date_And_Time = PLC DB302_InputDados.SKD.Turnos.2_Turno.Inicio AT %DB302.DBX384.0, 1 s
   "DB302_InputDados_SKD_Turnos_2_Turno_Fim" : Date_And_Time = PLC DB302_InputDados.SKD.Turnos.2_Turno.Fim AT %DB302.DBX392.0, 1 s
   "DB302_InputDados_SKD_Turnos_2_Turno_TempoTakt" : Int = PLC DB302_InputDados.SKD.Turnos.2_Turno.TempoTakt AT %DB302.DBW400, 1 s
   "DB302_InputDados_SKD_Turnos_2_Turno_Rodadas" : Int = PLC DB302_InputDados.SKD.Turnos.2_Turno.Rodadas AT %DB302.DBW402, 1 s
   "DB302_InputDados_SKD_Turnos_3_Turno_Inicio" : Date_And_Time = PLC DB302_InputDados.SKD.Turnos.3_Turno.Inicio AT %DB302.DBX404.0, 1 s
   "DB302_InputDados_SKD_Turnos_3_Turno_Fim" : Date_And_Time = PLC DB302_InputDados.SKD.Turnos.3_Turno.Fim AT %DB302.DBX412.0, 1 s
   "DB302_InputDados_SKD_Turnos_3_Turno_TempoTakt" : Int = PLC DB302_InputDados.SKD.Turnos.3_Turno.TempoTakt AT %DB302.DBW420, 1 s
   "DB302_InputDados_SKD_Turnos_3_Turno_Rodadas" : Int = PLC DB302_InputDados.SKD.Turnos.3_Turno.Rodadas AT %DB302.DBW422, 1 s
   "DB302_InputDados_SKD_SistemaOn" : Bool = PLC DB302_InputDados.SKD.SistemaOn AT %DB302.DBX544.0, 1 s
   "DB302_InputDados_Componentes_Turnos_1_Turno_Inicio" : Date_And_Time = PLC DB302_InputDados.Componentes.Turnos.1_Turno.Inicio AT %DB302.DBX546.0, 1 s
   "DB302_InputDados_Componentes_Turnos_1_Turno_Fim" : Date_And_Time = PLC DB302_InputDados.Componentes.Turnos.1_Turno.Fim AT %DB302.DBX554.0, 1 s
   "DB302_InputDados_Componentes_Turnos_1_Turno_TempoTakt" : Int = PLC DB302_InputDados.Componentes.Turnos.1_Turno.TempoTakt AT %DB302.DBW562, 1 s
   "DB302_InputDados_Componentes_Turnos_1_Turno_Rodadas" : Int = PLC DB302_InputDados.Componentes.Turnos.1_Turno.Rodadas AT %DB302.DBW564, 1 s
   "DB302_InputDados_Componentes_Turnos_2_Turno_Inicio" : Date_And_Time = PLC DB302_InputDados.Componentes.Turnos.2_Turno.Inicio AT %DB302.DBX566.0, 1 s
   "DB302_InputDados_Componentes_Turnos_2_Turno_Fim" : Date_And_Time = PLC DB302_InputDados.Componentes.Turnos.2_Turno.Fim AT %DB302.DBX574.0, 1 s
   "DB302_InputDados_Componentes_Turnos_2_Turno_TempoTakt" : Int = PLC DB302_InputDados.Componentes.Turnos.2_Turno.TempoTakt AT %DB302.DBW582, 1 s
   "DB302_InputDados_Componentes_Turnos_2_Turno_Rodadas" : Int = PLC DB302_InputDados.Componentes.Turnos.2_Turno.Rodadas AT %DB302.DBW584, 1 s
   "DB302_InputDados_Componentes_Turnos_3_Turno_Inicio" : Date_And_Time = PLC DB302_InputDados.Componentes.Turnos.3_Turno.Inicio AT %DB302.DBX586.0, 1 s
   "DB302_InputDados_Componentes_Turnos_3_Turno_Fim" : Date_And_Time = PLC DB302_InputDados.Componentes.Turnos.3_Turno.Fim AT %DB302.DBX594.0, 1 s
   "DB302_InputDados_Componentes_Turnos_3_Turno_TempoTakt" : Int = PLC DB302_InputDados.Componentes.Turnos.3_Turno.TempoTakt AT %DB302.DBW602, 1 s
   "DB302_InputDados_Componentes_Turnos_3_Turno_Rodadas" : Int = PLC DB302_InputDados.Componentes.Turnos.3_Turno.Rodadas AT %DB302.DBW604, 1 s
   "DB302_InputDados_Componentes_SistemaOn" : Bool = PLC DB302_InputDados.Componentes.SistemaOn AT %DB302.DBX726.0, 1 s
   "DB303_ScadaToCentral_Data_Turnos_Inicio{0}" : Time_Of_Day = PLC DB303_ScadaToCentral.Data.Turnos.Inicio[0] AT %DB303.DBD0, 1 s
   "DB303_ScadaToCentral_Data_Turnos_Fim{0}" : Time_Of_Day = PLC DB303_ScadaToCentral.Data.Turnos.Fim[0] AT %DB303.DBD12, 1 s
   "DB303_ScadaToCentral_Data_ParametrosTakt{0}_Tempo_Takt" : Int = PLC DB303_ScadaToCentral.Data.ParametrosTakt[0].Tempo_Takt AT %DB303.DBW74, 1 s
   "DB303_ScadaToCentral_Data_ParametrosTakt{0}_ObjetivoTurno" : Int = PLC DB303_ScadaToCentral.Data.ParametrosTakt[0].ObjetivoTurno AT %DB303.DBW76, 1 s
   "DB303_ScadaToCentral_Data_Turnos_Inicio{1}" : Time_Of_Day = PLC DB303_ScadaToCentral.Data.Turnos.Inicio[1] AT %DB303.DBD4, 1 s
   "DB303_ScadaToCentral_Data_Turnos_Fim{1}" : Time_Of_Day = PLC DB303_ScadaToCentral.Data.Turnos.Fim[1] AT %DB303.DBD16, 1 s
   "DB303_ScadaToCentral_Data_ParametrosTakt{1}_Tempo_Takt" : Int = PLC DB303_ScadaToCentral.Data.ParametrosTakt[1].Tempo_Takt AT %DB303.DBW78, 1 s
   "DB303_ScadaToCentral_Data_ParametrosTakt{1}_ObjetivoTurno" : Int = PLC DB303_ScadaToCentral.Data.ParametrosTakt[1].ObjetivoTurno AT %DB303.DBW80, 1 s
   "DB303_ScadaToCentral_Data_Turnos_Inicio{2}" : Time_Of_Day = PLC DB303_ScadaToCentral.Data.Turnos.Inicio[2] AT %DB303.DBD8, 1 s
   "DB303_ScadaToCentral_Data_Turnos_Fim{2}" : Time_Of_Day = PLC DB303_ScadaToCentral.Data.Turnos.Fim[2] AT %DB303.DBD20, 1 s
   "DB303_ScadaToCentral_Data_ParametrosTakt{2}_Tempo_Takt" : Int = PLC DB303_ScadaToCentral.Data.ParametrosTakt[2].Tempo_Takt AT %DB303.DBW82, 1 s
   "DB303_ScadaToCentral_Data_ParametrosTakt{2}_ObjetivoTurno" : Int = PLC DB303_ScadaToCentral.Data.ParametrosTakt[2].ObjetivoTurno AT %DB303.DBW84, 1 s
   "DB303_ScadaToCentral_Data_Dias_Da_Semana{0}" : Bool = PLC DB303_ScadaToCentral.Data.Dias_Da_Semana[0] AT %DB303.DBX72.0, 1 s
   "DB303_ScadaToCentral_Data_Dias_Da_Semana{1}" : Bool = PLC DB303_ScadaToCentral.Data.Dias_Da_Semana[1] AT %DB303.DBX72.1, 1 s
   "DB303_ScadaToCentral_Data_Dias_Da_Semana{2}" : Bool = PLC DB303_ScadaToCentral.Data.Dias_Da_Semana[2] AT %DB303.DBX72.2, 1 s
   "DB303_ScadaToCentral_Data_Dias_Da_Semana{3}" : Bool = PLC DB303_ScadaToCentral.Data.Dias_Da_Semana[3] AT %DB303.DBX72.3, 1 s
   "DB303_ScadaToCentral_Data_Dias_Da_Semana{4}" : Bool = PLC DB303_ScadaToCentral.Data.Dias_Da_Semana[4] AT %DB303.DBX72.4, 1 s
   "DB303_ScadaToCentral_Data_Dias_Da_Semana{5}" : Bool = PLC DB303_ScadaToCentral.Data.Dias_Da_Semana[5] AT %DB303.DBX72.5, 1 s
   "DB303_ScadaToCentral_Data_Dias_Da_Semana{6}" : Bool = PLC DB303_ScadaToCentral.Data.Dias_Da_Semana[6] AT %DB303.DBX72.6, 1 s
   "DB303_ScadaToCentral_Data_Paradas_Programadas_Inicio{0}" : Time_Of_Day = PLC DB303_ScadaToCentral.Data.Paradas_Programadas.Inicio[0] AT %DB303.DBD24, 1 s
   "DB303_ScadaToCentral_Data_Paradas_Programadas_Fim{0}" : Time_Of_Day = PLC DB303_ScadaToCentral.Data.Paradas_Programadas.Fim[0] AT %DB303.DBD48, 1 s
   "DB303_ScadaToCentral_Data_Paradas_Programadas_Inicio{1}" : Time_Of_Day = PLC DB303_ScadaToCentral.Data.Paradas_Programadas.Inicio[1] AT %DB303.DBD28, 1 s
   "DB303_ScadaToCentral_Data_Paradas_Programadas_Fim{1}" : Time_Of_Day = PLC DB303_ScadaToCentral.Data.Paradas_Programadas.Fim[1] AT %DB303.DBD52, 1 s
   "DB303_ScadaToCentral_Data_Paradas_Programadas_Inicio{2}" : Time_Of_Day = PLC DB303_ScadaToCentral.Data.Paradas_Programadas.Inicio[2] AT %DB303.DBD32, 1 s
   "DB303_ScadaToCentral_Data_Paradas_Programadas_Fim{2}" : Time_Of_Day = PLC DB303_ScadaToCentral.Data.Paradas_Programadas.Fim[2] AT %DB303.DBD56, 1 s
   "DB303_ScadaToCentral_Data_Paradas_Programadas_Inicio{4}" : Time_Of_Day = PLC DB303_ScadaToCentral.Data.Paradas_Programadas.Inicio[4] AT %DB303.DBD40, 1 s
   "DB303_ScadaToCentral_Data_Paradas_Programadas_Fim{5}" : Time_Of_Day = PLC DB303_ScadaToCentral.Data.Paradas_Programadas.Fim[5] AT %DB303.DBD68, 1 s
   "DB303_ScadaToCentral_Data_Paradas_Programadas_Fim{4}" : Time_Of_Day = PLC DB303_ScadaToCentral.Data.Paradas_Programadas.Fim[4] AT %DB303.DBD64, 1 s
   "DB303_ScadaToCentral_Data_Paradas_Programadas_Inicio{5}" : Time_Of_Day = PLC DB303_ScadaToCentral.Data.Paradas_Programadas.Inicio[5] AT %DB303.DBD44, 1 s

text list "Text_list_1": 0 'TAKT DESLIGADO'; 1 'TAKT LIGADO'

graphic list "@DiagnosticsStates": 0 '@Diagnostics_StateGood'; 1 '@Diagnostics_StateBad'

screen "01_PainelCab" 800x447
   Rectangle "Rectangle_9" at 1,2 size 798x443
      Appearance <- "DB300_IhmDados_Dados_Cabinas_CorDeTela"
   Rectangle "Rectangle_1" at 106,11 size 60x50
      Appearance <- "DB300_IhmDados_Dados_Cabinas_Andons{0}"
   TextField "Text field_1" at 129,27 size 14x20; Text '1'
   IOField "I/O field_3" at 84,74 size 156x40; FormatPattern 999999
      ProcessValue <- "DB300_IhmDados_Dados_Cabinas_Tempo_StopTime"
   TextField "Text field_4" at 52,198 size 249x29; Text 'OBJETIVO DO TURNO'
   Rectangle "Rectangle_2" at 175,11 size 60x50
      Appearance <- "DB300_IhmDados_Dados_Cabinas_Andons{1}"
   Rectangle "Rectangle_3" at 249,11 size 60x50
      Appearance <- "DB300_IhmDados_Dados_Cabinas_Andons{2}"
   Rectangle "Rectangle_4" at 322,11 size 60x50
      Appearance <- "DB300_IhmDados_Dados_Cabinas_Andons{3}"
   Rectangle "Rectangle_5" at 393,11 size 60x50
      Appearance <- "DB300_IhmDados_Dados_Cabinas_Andons{4}"
   Rectangle "Rectangle_6" at 465,12 size 60x50
      Appearance <- "DB300_IhmDados_Dados_Cabinas_Andons{5}"
   Rectangle "Rectangle_7" at 538,12 size 60x50
      Appearance <- "DB300_IhmDados_Dados_Cabinas_Andons{6}"
   TextField "Text field_6" at 198,27 size 14x20; Text '2'
   TextField "Text field_7" at 272,27 size 14x20; Text '3'
   TextField "Text field_8" at 344,27 size 14x20; Text '4'
   TextField "Text field_9" at 417,27 size 14x20; Text '5'
   TextField "Text field_10" at 490,27 size 14x20; Text '6'
   TextField "Text field_11" at 561,27 size 14x20; Text '7'
   Rectangle "Rectangle_8" at 607,12 size 60x50
      Appearance <- "DB300_IhmDados_Dados_Cabinas_Andons{7}"
   TextField "Text field_12" at 629,27 size 14x20; Text '8'
   IOField "I/O field_1" at 530,75 size 149x40; FormatPattern 999999
      ProcessValue <- "DB300_IhmDados_Dados_Cabinas_Tempo_Takt"
   TextField "Text field_2" at 571,119 size 80x29; Text 'TIMER'
   IOField "I/O field_4" at 561,160 size 93x40; FormatPattern 999
      ProcessValue <- "DB300_IhmDados_Dados_Cabinas_Atual"
   TextField "Text field_5" at 466,200 size 334x29; Text 'PRODUÇÃO ATÉ O MOMENTO'
   IOField "I/O field_5" at 562,236 size 93x40; FormatPattern 999
      ProcessValue <- "DB300_IhmDados_Dados_Cabinas_SaldoDoTurno"
   TextField "Text field_14" at 515,282 size 210x29; Text 'SALDO DO TURNO'
   IOField "I/O field_6" at 119,236 size 93x40; FormatPattern 99.9
      ProcessValue <- "DB300_IhmDados_Dados_Cabinas_DirectRun"
   TextField "Text field_15" at 91,276 size 149x29; Text 'DIRECT RUN'
   IOField "I/O field_2" at 120,158 size 93x40; FormatPattern 999
      ProcessValue <- "DB300_IhmDados_Dados_Cabinas_Objetivo"
   TextField "Text field_3" at 101,119 size 131x29; Text 'STOP TIME'
   IOField "I/O field_7" at 2,356 size 794x75; FormatPattern ????????????????????????????????????????????????????????????????????????????????
      ProcessValue <- "DB300_IhmDados_Mensagem_Cab"
   Button "Button_1" at 7,19 size 88x30; TextOff 'HOME'
      on Release: ActivateScreen("01_Home", 0)

screen "01_PainelComp" 800x447
   Rectangle "Rectangle_9" at 1,2 size 798x443
      Appearance <- "DB300_IhmDados_Dados_Componentes_CorDeTela"
   Rectangle "Rectangle_1" at 106,11 size 60x50
      Appearance <- "DB300_IhmDados_Dados_Componentes_Andons{0}"
   TextField "Text field_1" at 129,27 size 14x20; Text '1'
   IOField "I/O field_3" at 84,74 size 156x40; FormatPattern 999999
      ProcessValue <- "DB300_IhmDados_Dados_Componentes_Tempo_StopTime"
   TextField "Text field_4" at 52,198 size 249x29; Text 'OBJETIVO DO TURNO'
   Rectangle "Rectangle_2" at 175,11 size 60x50
      Appearance <- "DB300_IhmDados_Dados_Componentes_Andons{1}"
   Rectangle "Rectangle_3" at 249,11 size 60x50
      Appearance <- "DB300_IhmDados_Dados_Componentes_Andons{2}"
   Rectangle "Rectangle_4" at 322,11 size 60x50
      Appearance <- "DB300_IhmDados_Dados_Componentes_Andons{3}"
   Rectangle "Rectangle_5" at 393,11 size 60x50
      Appearance <- "DB300_IhmDados_Dados_Componentes_Andons{4}"
   Rectangle "Rectangle_6" at 465,12 size 60x50
      Appearance <- "DB300_IhmDados_Dados_Componentes_Andons{5}"
   Rectangle "Rectangle_7" at 538,12 size 60x50
      Appearance <- "DB300_IhmDados_Dados_Componentes_Andons{6}"
   TextField "Text field_6" at 198,27 size 14x20; Text '2'
   TextField "Text field_7" at 272,27 size 14x20; Text '3'
   TextField "Text field_8" at 344,27 size 14x20; Text '4'
   TextField "Text field_9" at 417,27 size 14x20; Text '5'
   TextField "Text field_10" at 490,27 size 14x20; Text '6'
   TextField "Text field_11" at 561,27 size 14x20; Text '7'
   Rectangle "Rectangle_8" at 607,12 size 60x50
      Appearance <- "DB300_IhmDados_Dados_Componentes_Andons{7}"
   TextField "Text field_12" at 629,27 size 14x20; Text '8'
   IOField "I/O field_1" at 530,75 size 149x40; FormatPattern 999999
      ProcessValue <- "DB300_IhmDados_Dados_Componentes_Tempo_Takt"
   TextField "Text field_2" at 571,119 size 80x29; Text 'TIMER'
   IOField "I/O field_4" at 561,160 size 93x40; FormatPattern 999
      ProcessValue <- "DB300_IhmDados_Dados_Componentes_Atual"
   TextField "Text field_5" at 466,200 size 334x29; Text 'PRODUÇÃO ATÉ O MOMENTO'
   IOField "I/O field_5" at 562,236 size 93x40; FormatPattern 999
      ProcessValue <- "DB300_IhmDados_Dados_Componentes_SaldoDoTurno"
   TextField "Text field_14" at 515,282 size 210x29; Text 'SALDO DO TURNO'
   IOField "I/O field_6" at 119,236 size 93x40; FormatPattern 99.9
      ProcessValue <- "DB300_IhmDados_Dados_Componentes_DirectRun"
   TextField "Text field_15" at 91,276 size 149x29; Text 'DIRECT RUN'
   IOField "I/O field_2" at 120,158 size 93x40; FormatPattern 999
      ProcessValue <- "DB300_IhmDados_Dados_Componentes_Objetivo"
   TextField "Text field_3" at 101,119 size 131x29; Text 'STOP TIME'
   IOField "I/O field_7" at 2,356 size 794x75; FormatPattern ????????????????????????????????????????????????????????????????????????????????
      ProcessValue <- "DB300_IhmDados_Mensagem_Componentes"
   Button "Button_1" at 7,19 size 88x30; TextOff 'HOME'
      on Release: ActivateScreen("01_Home", 0)

screen "01_PainelSkd" 800x447
   Rectangle "Rectangle_9" at 1,2 size 798x443
      Appearance <- "DB300_IhmDados_Dados_SKD_CorDeTela"
   Rectangle "Rectangle_1" at 106,11 size 60x50
      Appearance <- "DB300_IhmDados_Dados_SKD_Andons{0}"
   TextField "Text field_1" at 129,27 size 14x20; Text '1'
   IOField "I/O field_3" at 84,74 size 156x40; FormatPattern 999999
      ProcessValue <- "DB300_IhmDados_Dados_SKD_Tempo_StopTime"
   TextField "Text field_4" at 52,198 size 249x29; Text 'OBJETIVO DO TURNO'
   Rectangle "Rectangle_2" at 175,11 size 60x50
      Appearance <- "DB300_IhmDados_Dados_SKD_Andons{1}"
   Rectangle "Rectangle_3" at 249,11 size 60x50
      Appearance <- "DB300_IhmDados_Dados_SKD_Andons{2}"
   Rectangle "Rectangle_4" at 322,11 size 60x50
      Appearance <- "DB300_IhmDados_Dados_SKD_Andons{3}"
   Rectangle "Rectangle_5" at 393,11 size 60x50
      Appearance <- "DB300_IhmDados_Dados_SKD_Andons{4}"
   Rectangle "Rectangle_6" at 465,12 size 60x50
      Appearance <- "DB300_IhmDados_Dados_SKD_Andons{5}"
   Rectangle "Rectangle_7" at 538,12 size 60x50
      Appearance <- "DB300_IhmDados_Dados_SKD_Andons{6}"
   TextField "Text field_6" at 198,27 size 14x20; Text '2'
   TextField "Text field_7" at 272,27 size 14x20; Text '3'
   TextField "Text field_8" at 344,27 size 14x20; Text '4'
   TextField "Text field_9" at 417,27 size 14x20; Text '5'
   TextField "Text field_10" at 490,27 size 14x20; Text '6'
   TextField "Text field_11" at 561,27 size 14x20; Text '7'
   Rectangle "Rectangle_8" at 607,12 size 60x50
      Appearance <- "DB300_IhmDados_Dados_SKD_Andons{7}"
   TextField "Text field_12" at 629,27 size 14x20; Text '8'
   IOField "I/O field_1" at 530,75 size 149x40; FormatPattern 999999
      ProcessValue <- "DB300_IhmDados_Dados_SKD_Tempo_Takt"
   TextField "Text field_2" at 571,119 size 80x29; Text 'TIMER'
   IOField "I/O field_4" at 561,160 size 93x40; FormatPattern 999
      ProcessValue <- "DB300_IhmDados_Dados_SKD_Atual"
   TextField "Text field_5" at 466,200 size 334x29; Text 'PRODUÇÃO ATÉ O MOMENTO'
   IOField "I/O field_5" at 562,236 size 93x40; FormatPattern 999
      ProcessValue <- "DB300_IhmDados_Dados_SKD_SaldoDoTurno"
   TextField "Text field_14" at 515,282 size 210x29; Text 'SALDO DO TURNO'
   IOField "I/O field_6" at 119,236 size 93x40; FormatPattern 99.9
      ProcessValue <- "DB300_IhmDados_Dados_SKD_DirectRun"
   TextField "Text field_15" at 91,276 size 149x29; Text 'DIRECT RUN'
   IOField "I/O field_2" at 120,158 size 93x40; FormatPattern 999
      ProcessValue <- "DB300_IhmDados_Dados_SKD_Objetivo"
   TextField "Text field_3" at 101,119 size 131x29; Text 'STOP TIME'
   IOField "I/O field_7" at 2,356 size 794x75; FormatPattern ????????????????????????????????????????????????????????????????????????????????
      ProcessValue <- "DB300_IhmDados_Mensagem_SKD"
   Button "Button_1" at 7,19 size 88x30; TextOff 'HOME'
      on Release: ActivateScreen("01_Home", 0)

screen "01_PainelEcu" 800x447
   Rectangle "Rectangle_9" at 1,2 size 798x443
      Appearance <- "DB300_IhmDados_Dados_ECU_CorDeTela"
   Rectangle "Rectangle_1" at 106,11 size 60x50
      Appearance <- "DB300_IhmDados_Dados_ECU_Andons{0}"
   TextField "Text field_1" at 129,27 size 14x20; Text '1'
   IOField "I/O field_3" at 84,74 size 156x40; FormatPattern 999999
      ProcessValue <- "DB300_IhmDados_Dados_ECU_Tempo_StopTime"
   TextField "Text field_4" at 52,198 size 249x29; Text 'OBJETIVO DO TURNO'
   Rectangle "Rectangle_2" at 175,11 size 60x50
      Appearance <- "DB300_IhmDados_Dados_ECU_Andons{1}"
   Rectangle "Rectangle_3" at 249,11 size 60x50
      Appearance <- "DB300_IhmDados_Dados_ECU_Andons{2}"
   Rectangle "Rectangle_4" at 322,11 size 60x50
      Appearance <- "DB300_IhmDados_Dados_ECU_Andons{3}"
   Rectangle "Rectangle_5" at 393,11 size 60x50
      Appearance <- "DB300_IhmDados_Dados_ECU_Andons{4}"
   Rectangle "Rectangle_6" at 465,12 size 60x50
      Appearance <- "DB300_IhmDados_Dados_ECU_Andons{5}"
   Rectangle "Rectangle_7" at 538,12 size 60x50
      Appearance <- "DB300_IhmDados_Dados_ECU_Andons{6}"
   TextField "Text field_6" at 198,27 size 14x20; Text '2'
   TextField "Text field_7" at 272,27 size 14x20; Text '3'
   TextField "Text field_8" at 344,27 size 14x20; Text '4'
   TextField "Text field_9" at 417,27 size 14x20; Text '5'
   TextField "Text field_10" at 490,27 size 14x20; Text '6'
   TextField "Text field_11" at 561,27 size 14x20; Text '7'
   Rectangle "Rectangle_8" at 607,12 size 60x50
      Appearance <- "DB300_IhmDados_Dados_ECU_Andons{7}"
   TextField "Text field_12" at 629,27 size 14x20; Text '8'
   IOField "I/O field_1" at 530,75 size 149x40; FormatPattern 999999
      ProcessValue <- "DB300_IhmDados_Dados_ECU_Tempo_Takt"
   TextField "Text field_2" at 571,119 size 80x29; Text 'TIMER'
   IOField "I/O field_4" at 561,160 size 93x40; FormatPattern 999
      ProcessValue <- "DB300_IhmDados_Dados_ECU_Atual"
   TextField "Text field_5" at 466,200 size 334x29; Text 'PRODUÇÃO ATÉ O MOMENTO'
   IOField "I/O field_5" at 562,236 size 93x40; FormatPattern 999
      ProcessValue <- "DB300_IhmDados_Dados_ECU_SaldoDoTurno"
   TextField "Text field_14" at 515,282 size 210x29; Text 'SALDO DO TURNO'
   IOField "I/O field_6" at 119,236 size 93x40; FormatPattern 99.9
      ProcessValue <- "DB300_IhmDados_Dados_ECU_DirectRun"
   TextField "Text field_15" at 91,276 size 149x29; Text 'DIRECT RUN'
   IOField "I/O field_2" at 120,158 size 93x40; FormatPattern 999
      ProcessValue <- "DB300_IhmDados_Dados_ECU_Objetivo"
   TextField "Text field_3" at 101,119 size 131x29; Text 'STOP TIME'
   IOField "I/O field_7" at 2,356 size 794x75; FormatPattern ????????????????????????????????????????????????????????????????????????????????
      ProcessValue <- "DB300_IhmDados_Mensagem_ECU"
   Button "Button_1" at 7,19 size 88x30; TextOff 'HOME'
      on Release: ActivateScreen("01_Home", 0)

screen "01_Home" 800x447, template "Template_1"
   Button "Button_1" at 25,365 size 181x32; TextOff 'PAINEL CABINAS'
      on Release: ActivateScreen("01_PainelCab", 0)
   Button "Button_2" at 209,365 size 181x32; TextOff 'PAINEL SKD'
      on Release: ActivateScreen("01_PainelSkd", 0)
   Button "Button_3" at 393,365 size 181x32; TextOff 'PAINEL COMPONENTES'
      on Release: ActivateScreen("01_PainelComp", 0)
   Button "Button_4" at 577,365 size 181x32; TextOff 'PAINEL ECU'
      on Release: ActivateScreen("01_PainelEcu", 0)
   Button "Button_5" at 26,410 size 181x32; TextOff 'PARAMETROS CABINAS'
      on Release: ActivateScreen("02_Parametros_Cab", 0)
   Button "Button_6" at 577,410 size 181x32; TextOff 'PARAMETROS ECU'
      on Release: ActivateScreen("02_Parametros_Ecu", 0)
   Button "Button_7" at 393,410 size 181x32; TextOff 'PARAMETROS COMP.'
      on Release: ActivateScreen("02_Parametros_Comp", 0)
   Button "Button_8" at 209,410 size 181x32; TextOff 'PARAMETROS SKD'
      on Release: ActivateScreen("02_Parametros_Skd", 0)

